   // GBK_TO_UNICODE[22068] := 16#C29A;
   // GBK_TO_UNICODE[22069] := 16#8077;
   // GBK_TO_UNICODE[22070] := 16#C29B;
   // GBK_TO_UNICODE[22071] := 16#8078;
   // GBK_TO_UNICODE[22072] := 16#C29C;
   // GBK_TO_UNICODE[22073] := 16#8079;
   // GBK_TO_UNICODE[22074] := 16#C29D;
   // GBK_TO_UNICODE[22075] := 16#807A;
   // GBK_TO_UNICODE[22076] := 16#C29E;
   // GBK_TO_UNICODE[22077] := 16#807B;
   // GBK_TO_UNICODE[22078] := 16#C29F;
   // GBK_TO_UNICODE[22079] := 16#807C;
   // GBK_TO_UNICODE[22080] := 16#C2A0;
   // GBK_TO_UNICODE[22081] := 16#807D;
   // GBK_TO_UNICODE[22082] := 16#C2A1;
   // GBK_TO_UNICODE[22083] := 16#9686;
   // GBK_TO_UNICODE[22084] := 16#C2A2;
   // GBK_TO_UNICODE[22085] := 16#5784;
   // GBK_TO_UNICODE[22086] := 16#C2A3;
   // GBK_TO_UNICODE[22087] := 16#62E2;
   // GBK_TO_UNICODE[22088] := 16#C2A4;
   // GBK_TO_UNICODE[22089] := 16#9647;
   // GBK_TO_UNICODE[22090] := 16#C2A5;
   // GBK_TO_UNICODE[22091] := 16#697C;
   // GBK_TO_UNICODE[22092] := 16#C2A6;
   // GBK_TO_UNICODE[22093] := 16#5A04;
   // GBK_TO_UNICODE[22094] := 16#C2A7;
   // GBK_TO_UNICODE[22095] := 16#6402;
   // GBK_TO_UNICODE[22096] := 16#C2A8;
   // GBK_TO_UNICODE[22097] := 16#7BD3;
   // GBK_TO_UNICODE[22098] := 16#C2A9;
   // GBK_TO_UNICODE[22099] := 16#6F0F;
   // GBK_TO_UNICODE[22100] := 16#C2AA;
   // GBK_TO_UNICODE[22101] := 16#964B;
   // GBK_TO_UNICODE[22102] := 16#C2AB;
   // GBK_TO_UNICODE[22103] := 16#82A6;
   // GBK_TO_UNICODE[22104] := 16#C2AC;
   // GBK_TO_UNICODE[22105] := 16#5362;
   // GBK_TO_UNICODE[22106] := 16#C2AD;
   // GBK_TO_UNICODE[22107] := 16#9885;
   // GBK_TO_UNICODE[22108] := 16#C2AE;
   // GBK_TO_UNICODE[22109] := 16#5E90;
   // GBK_TO_UNICODE[22110] := 16#C2AF;
   // GBK_TO_UNICODE[22111] := 16#7089;
   // GBK_TO_UNICODE[22112] := 16#C2B0;
   // GBK_TO_UNICODE[22113] := 16#63B3;
   // GBK_TO_UNICODE[22114] := 16#C2B1;
   // GBK_TO_UNICODE[22115] := 16#5364;
   // GBK_TO_UNICODE[22116] := 16#C2B2;
   // GBK_TO_UNICODE[22117] := 16#864F;
   // GBK_TO_UNICODE[22118] := 16#C2B3;
   // GBK_TO_UNICODE[22119] := 16#9C81;
   // GBK_TO_UNICODE[22120] := 16#C2B4;
   // GBK_TO_UNICODE[22121] := 16#9E93;
   // GBK_TO_UNICODE[22122] := 16#C2B5;
   // GBK_TO_UNICODE[22123] := 16#788C;
   // GBK_TO_UNICODE[22124] := 16#C2B6;
   // GBK_TO_UNICODE[22125] := 16#9732;
   // GBK_TO_UNICODE[22126] := 16#C2B7;
   // GBK_TO_UNICODE[22127] := 16#8DEF;
   // GBK_TO_UNICODE[22128] := 16#C2B8;
   // GBK_TO_UNICODE[22129] := 16#8D42;
   // GBK_TO_UNICODE[22130] := 16#C2B9;
   // GBK_TO_UNICODE[22131] := 16#9E7F;
   // GBK_TO_UNICODE[22132] := 16#C2BA;
   // GBK_TO_UNICODE[22133] := 16#6F5E;
   // GBK_TO_UNICODE[22134] := 16#C2BB;
   // GBK_TO_UNICODE[22135] := 16#7984;
   // GBK_TO_UNICODE[22136] := 16#C2BC;
   // GBK_TO_UNICODE[22137] := 16#5F55;
   // GBK_TO_UNICODE[22138] := 16#C2BD;
   // GBK_TO_UNICODE[22139] := 16#9646;
   // GBK_TO_UNICODE[22140] := 16#C2BE;
   // GBK_TO_UNICODE[22141] := 16#622E;
   // GBK_TO_UNICODE[22142] := 16#C2BF;
   // GBK_TO_UNICODE[22143] := 16#9A74;
   // GBK_TO_UNICODE[22144] := 16#C2C0;
   // GBK_TO_UNICODE[22145] := 16#5415;
   // GBK_TO_UNICODE[22146] := 16#C2C1;
   // GBK_TO_UNICODE[22147] := 16#94DD;
   // GBK_TO_UNICODE[22148] := 16#C2C2;
   // GBK_TO_UNICODE[22149] := 16#4FA3;
   // GBK_TO_UNICODE[22150] := 16#C2C3;
   // GBK_TO_UNICODE[22151] := 16#65C5;
   // GBK_TO_UNICODE[22152] := 16#C2C4;
   // GBK_TO_UNICODE[22153] := 16#5C65;
   // GBK_TO_UNICODE[22154] := 16#C2C5;
   // GBK_TO_UNICODE[22155] := 16#5C61;
   // GBK_TO_UNICODE[22156] := 16#C2C6;
   // GBK_TO_UNICODE[22157] := 16#7F15;
   // GBK_TO_UNICODE[22158] := 16#C2C7;
   // GBK_TO_UNICODE[22159] := 16#8651;
   // GBK_TO_UNICODE[22160] := 16#C2C8;
   // GBK_TO_UNICODE[22161] := 16#6C2F;
   // GBK_TO_UNICODE[22162] := 16#C2C9;
   // GBK_TO_UNICODE[22163] := 16#5F8B;
   // GBK_TO_UNICODE[22164] := 16#C2CA;
   // GBK_TO_UNICODE[22165] := 16#7387;
   // GBK_TO_UNICODE[22166] := 16#C2CB;
   // GBK_TO_UNICODE[22167] := 16#6EE4;
   // GBK_TO_UNICODE[22168] := 16#C2CC;
   // GBK_TO_UNICODE[22169] := 16#7EFF;
   // GBK_TO_UNICODE[22170] := 16#C2CD;
   // GBK_TO_UNICODE[22171] := 16#5CE6;
   // GBK_TO_UNICODE[22172] := 16#C2CE;
   // GBK_TO_UNICODE[22173] := 16#631B;
   // GBK_TO_UNICODE[22174] := 16#C2CF;
   // GBK_TO_UNICODE[22175] := 16#5B6A;
   // GBK_TO_UNICODE[22176] := 16#C2D0;
   // GBK_TO_UNICODE[22177] := 16#6EE6;
   // GBK_TO_UNICODE[22178] := 16#C2D1;
   // GBK_TO_UNICODE[22179] := 16#5375;
   // GBK_TO_UNICODE[22180] := 16#C2D2;
   // GBK_TO_UNICODE[22181] := 16#4E71;
   // GBK_TO_UNICODE[22182] := 16#C2D3;
   // GBK_TO_UNICODE[22183] := 16#63A0;
   // GBK_TO_UNICODE[22184] := 16#C2D4;
   // GBK_TO_UNICODE[22185] := 16#7565;
   // GBK_TO_UNICODE[22186] := 16#C2D5;
   // GBK_TO_UNICODE[22187] := 16#62A1;
   // GBK_TO_UNICODE[22188] := 16#C2D6;
   // GBK_TO_UNICODE[22189] := 16#8F6E;
   // GBK_TO_UNICODE[22190] := 16#C2D7;
   // GBK_TO_UNICODE[22191] := 16#4F26;
   // GBK_TO_UNICODE[22192] := 16#C2D8;
   // GBK_TO_UNICODE[22193] := 16#4ED1;
   // GBK_TO_UNICODE[22194] := 16#C2D9;
   // GBK_TO_UNICODE[22195] := 16#6CA6;
   // GBK_TO_UNICODE[22196] := 16#C2DA;
   // GBK_TO_UNICODE[22197] := 16#7EB6;
   // GBK_TO_UNICODE[22198] := 16#C2DB;
   // GBK_TO_UNICODE[22199] := 16#8BBA;
   // GBK_TO_UNICODE[22200] := 16#C2DC;
   // GBK_TO_UNICODE[22201] := 16#841D;
   // GBK_TO_UNICODE[22202] := 16#C2DD;
   // GBK_TO_UNICODE[22203] := 16#87BA;
   // GBK_TO_UNICODE[22204] := 16#C2DE;
   // GBK_TO_UNICODE[22205] := 16#7F57;
   // GBK_TO_UNICODE[22206] := 16#C2DF;
   // GBK_TO_UNICODE[22207] := 16#903B;
   // GBK_TO_UNICODE[22208] := 16#C2E0;
   // GBK_TO_UNICODE[22209] := 16#9523;
   // GBK_TO_UNICODE[22210] := 16#C2E1;
   // GBK_TO_UNICODE[22211] := 16#7BA9;
   // GBK_TO_UNICODE[22212] := 16#C2E2;
   // GBK_TO_UNICODE[22213] := 16#9AA1;
   // GBK_TO_UNICODE[22214] := 16#C2E3;
   // GBK_TO_UNICODE[22215] := 16#88F8;
   // GBK_TO_UNICODE[22216] := 16#C2E4;
   // GBK_TO_UNICODE[22217] := 16#843D;
   // GBK_TO_UNICODE[22218] := 16#C2E5;
   // GBK_TO_UNICODE[22219] := 16#6D1B;
   // GBK_TO_UNICODE[22220] := 16#C2E6;
   // GBK_TO_UNICODE[22221] := 16#9A86;
   // GBK_TO_UNICODE[22222] := 16#C2E7;
   // GBK_TO_UNICODE[22223] := 16#7EDC;
   // GBK_TO_UNICODE[22224] := 16#C2E8;
   // GBK_TO_UNICODE[22225] := 16#5988;
   // GBK_TO_UNICODE[22226] := 16#C2E9;
   // GBK_TO_UNICODE[22227] := 16#9EBB;
   // GBK_TO_UNICODE[22228] := 16#C2EA;
   // GBK_TO_UNICODE[22229] := 16#739B;
   // GBK_TO_UNICODE[22230] := 16#C2EB;
   // GBK_TO_UNICODE[22231] := 16#7801;
   // GBK_TO_UNICODE[22232] := 16#C2EC;
   // GBK_TO_UNICODE[22233] := 16#8682;
   // GBK_TO_UNICODE[22234] := 16#C2ED;
   // GBK_TO_UNICODE[22235] := 16#9A6C;
   // GBK_TO_UNICODE[22236] := 16#C2EE;
   // GBK_TO_UNICODE[22237] := 16#9A82;
   // GBK_TO_UNICODE[22238] := 16#C2EF;
   // GBK_TO_UNICODE[22239] := 16#561B;
   // GBK_TO_UNICODE[22240] := 16#C2F0;
   // GBK_TO_UNICODE[22241] := 16#5417;
   // GBK_TO_UNICODE[22242] := 16#C2F1;
   // GBK_TO_UNICODE[22243] := 16#57CB;
   // GBK_TO_UNICODE[22244] := 16#C2F2;
   // GBK_TO_UNICODE[22245] := 16#4E70;
   // GBK_TO_UNICODE[22246] := 16#C2F3;
   // GBK_TO_UNICODE[22247] := 16#9EA6;
   // GBK_TO_UNICODE[22248] := 16#C2F4;
   // GBK_TO_UNICODE[22249] := 16#5356;
   // GBK_TO_UNICODE[22250] := 16#C2F5;
   // GBK_TO_UNICODE[22251] := 16#8FC8;
   // GBK_TO_UNICODE[22252] := 16#C2F6;
   // GBK_TO_UNICODE[22253] := 16#8109;
   // GBK_TO_UNICODE[22254] := 16#C2F7;
   // GBK_TO_UNICODE[22255] := 16#7792;
   // GBK_TO_UNICODE[22256] := 16#C2F8;
   // GBK_TO_UNICODE[22257] := 16#9992;
   // GBK_TO_UNICODE[22258] := 16#C2F9;
   // GBK_TO_UNICODE[22259] := 16#86EE;
   // GBK_TO_UNICODE[22260] := 16#C2FA;
   // GBK_TO_UNICODE[22261] := 16#6EE1;
   // GBK_TO_UNICODE[22262] := 16#C2FB;
   // GBK_TO_UNICODE[22263] := 16#8513;
   // GBK_TO_UNICODE[22264] := 16#C2FC;
   // GBK_TO_UNICODE[22265] := 16#66FC;
   // GBK_TO_UNICODE[22266] := 16#C2FD;
   // GBK_TO_UNICODE[22267] := 16#6162;
   // GBK_TO_UNICODE[22268] := 16#C2FE;
   // GBK_TO_UNICODE[22269] := 16#6F2B;
   // GBK_TO_UNICODE[22270] := 16#C340;
   // GBK_TO_UNICODE[22271] := 16#807E;
   // GBK_TO_UNICODE[22272] := 16#C341;
   // GBK_TO_UNICODE[22273] := 16#8081;
   // GBK_TO_UNICODE[22274] := 16#C342;
   // GBK_TO_UNICODE[22275] := 16#8082;
   // GBK_TO_UNICODE[22276] := 16#C343;
   // GBK_TO_UNICODE[22277] := 16#8085;
   // GBK_TO_UNICODE[22278] := 16#C344;
   // GBK_TO_UNICODE[22279] := 16#8088;
   // GBK_TO_UNICODE[22280] := 16#C345;
   // GBK_TO_UNICODE[22281] := 16#808A;
   // GBK_TO_UNICODE[22282] := 16#C346;
   // GBK_TO_UNICODE[22283] := 16#808D;
   // GBK_TO_UNICODE[22284] := 16#C347;
   // GBK_TO_UNICODE[22285] := 16#808E;
   // GBK_TO_UNICODE[22286] := 16#C348;
   // GBK_TO_UNICODE[22287] := 16#808F;
   // GBK_TO_UNICODE[22288] := 16#C349;
   // GBK_TO_UNICODE[22289] := 16#8090;
   // GBK_TO_UNICODE[22290] := 16#C34A;
   // GBK_TO_UNICODE[22291] := 16#8091;
   // GBK_TO_UNICODE[22292] := 16#C34B;
   // GBK_TO_UNICODE[22293] := 16#8092;
   // GBK_TO_UNICODE[22294] := 16#C34C;
   // GBK_TO_UNICODE[22295] := 16#8094;
   // GBK_TO_UNICODE[22296] := 16#C34D;
   // GBK_TO_UNICODE[22297] := 16#8095;
   // GBK_TO_UNICODE[22298] := 16#C34E;
   // GBK_TO_UNICODE[22299] := 16#8097;
   // GBK_TO_UNICODE[22300] := 16#C34F;
   // GBK_TO_UNICODE[22301] := 16#8099;
   // GBK_TO_UNICODE[22302] := 16#C350;
   // GBK_TO_UNICODE[22303] := 16#809E;
   // GBK_TO_UNICODE[22304] := 16#C351;
   // GBK_TO_UNICODE[22305] := 16#80A3;
   // GBK_TO_UNICODE[22306] := 16#C352;
   // GBK_TO_UNICODE[22307] := 16#80A6;
   // GBK_TO_UNICODE[22308] := 16#C353;
   // GBK_TO_UNICODE[22309] := 16#80A7;
   // GBK_TO_UNICODE[22310] := 16#C354;
   // GBK_TO_UNICODE[22311] := 16#80A8;
   // GBK_TO_UNICODE[22312] := 16#C355;
   // GBK_TO_UNICODE[22313] := 16#80AC;
   // GBK_TO_UNICODE[22314] := 16#C356;
   // GBK_TO_UNICODE[22315] := 16#80B0;
   // GBK_TO_UNICODE[22316] := 16#C357;
   // GBK_TO_UNICODE[22317] := 16#80B3;
   // GBK_TO_UNICODE[22318] := 16#C358;
   // GBK_TO_UNICODE[22319] := 16#80B5;
   // GBK_TO_UNICODE[22320] := 16#C359;
   // GBK_TO_UNICODE[22321] := 16#80B6;
   // GBK_TO_UNICODE[22322] := 16#C35A;
   // GBK_TO_UNICODE[22323] := 16#80B8;
   // GBK_TO_UNICODE[22324] := 16#C35B;
   // GBK_TO_UNICODE[22325] := 16#80B9;
   // GBK_TO_UNICODE[22326] := 16#C35C;
   // GBK_TO_UNICODE[22327] := 16#80BB;
   // GBK_TO_UNICODE[22328] := 16#C35D;
   // GBK_TO_UNICODE[22329] := 16#80C5;
   // GBK_TO_UNICODE[22330] := 16#C35E;
   // GBK_TO_UNICODE[22331] := 16#80C7;
   // GBK_TO_UNICODE[22332] := 16#C35F;
   // GBK_TO_UNICODE[22333] := 16#80C8;
   // GBK_TO_UNICODE[22334] := 16#C360;
   // GBK_TO_UNICODE[22335] := 16#80C9;
   // GBK_TO_UNICODE[22336] := 16#C361;
   // GBK_TO_UNICODE[22337] := 16#80CA;
   // GBK_TO_UNICODE[22338] := 16#C362;
   // GBK_TO_UNICODE[22339] := 16#80CB;
   // GBK_TO_UNICODE[22340] := 16#C363;
   // GBK_TO_UNICODE[22341] := 16#80CF;
   // GBK_TO_UNICODE[22342] := 16#C364;
   // GBK_TO_UNICODE[22343] := 16#80D0;
   // GBK_TO_UNICODE[22344] := 16#C365;
   // GBK_TO_UNICODE[22345] := 16#80D1;
   // GBK_TO_UNICODE[22346] := 16#C366;
   // GBK_TO_UNICODE[22347] := 16#80D2;
   // GBK_TO_UNICODE[22348] := 16#C367;
   // GBK_TO_UNICODE[22349] := 16#80D3;
   // GBK_TO_UNICODE[22350] := 16#C368;
   // GBK_TO_UNICODE[22351] := 16#80D4;
   // GBK_TO_UNICODE[22352] := 16#C369;
   // GBK_TO_UNICODE[22353] := 16#80D5;
   // GBK_TO_UNICODE[22354] := 16#C36A;
   // GBK_TO_UNICODE[22355] := 16#80D8;
   // GBK_TO_UNICODE[22356] := 16#C36B;
   // GBK_TO_UNICODE[22357] := 16#80DF;
   // GBK_TO_UNICODE[22358] := 16#C36C;
   // GBK_TO_UNICODE[22359] := 16#80E0;
   // GBK_TO_UNICODE[22360] := 16#C36D;
   // GBK_TO_UNICODE[22361] := 16#80E2;
   // GBK_TO_UNICODE[22362] := 16#C36E;
   // GBK_TO_UNICODE[22363] := 16#80E3;
   // GBK_TO_UNICODE[22364] := 16#C36F;
   // GBK_TO_UNICODE[22365] := 16#80E6;
   // GBK_TO_UNICODE[22366] := 16#C370;
   // GBK_TO_UNICODE[22367] := 16#80EE;
   // GBK_TO_UNICODE[22368] := 16#C371;
   // GBK_TO_UNICODE[22369] := 16#80F5;
   // GBK_TO_UNICODE[22370] := 16#C372;
   // GBK_TO_UNICODE[22371] := 16#80F7;
   // GBK_TO_UNICODE[22372] := 16#C373;
   // GBK_TO_UNICODE[22373] := 16#80F9;
   // GBK_TO_UNICODE[22374] := 16#C374;
   // GBK_TO_UNICODE[22375] := 16#80FB;
   // GBK_TO_UNICODE[22376] := 16#C375;
   // GBK_TO_UNICODE[22377] := 16#80FE;
   // GBK_TO_UNICODE[22378] := 16#C376;
   // GBK_TO_UNICODE[22379] := 16#80FF;
   // GBK_TO_UNICODE[22380] := 16#C377;
   // GBK_TO_UNICODE[22381] := 16#8100;
   // GBK_TO_UNICODE[22382] := 16#C378;
   // GBK_TO_UNICODE[22383] := 16#8101;
   // GBK_TO_UNICODE[22384] := 16#C379;
   // GBK_TO_UNICODE[22385] := 16#8103;
   // GBK_TO_UNICODE[22386] := 16#C37A;
   // GBK_TO_UNICODE[22387] := 16#8104;
   // GBK_TO_UNICODE[22388] := 16#C37B;
   // GBK_TO_UNICODE[22389] := 16#8105;
   // GBK_TO_UNICODE[22390] := 16#C37C;
   // GBK_TO_UNICODE[22391] := 16#8107;
   // GBK_TO_UNICODE[22392] := 16#C37D;
   // GBK_TO_UNICODE[22393] := 16#8108;
   // GBK_TO_UNICODE[22394] := 16#C37E;
   // GBK_TO_UNICODE[22395] := 16#810B;
   // GBK_TO_UNICODE[22396] := 16#C380;
   // GBK_TO_UNICODE[22397] := 16#810C;
   // GBK_TO_UNICODE[22398] := 16#C381;
   // GBK_TO_UNICODE[22399] := 16#8115;
   // GBK_TO_UNICODE[22400] := 16#C382;
   // GBK_TO_UNICODE[22401] := 16#8117;
   // GBK_TO_UNICODE[22402] := 16#C383;
   // GBK_TO_UNICODE[22403] := 16#8119;
   // GBK_TO_UNICODE[22404] := 16#C384;
   // GBK_TO_UNICODE[22405] := 16#811B;
   // GBK_TO_UNICODE[22406] := 16#C385;
   // GBK_TO_UNICODE[22407] := 16#811C;
   // GBK_TO_UNICODE[22408] := 16#C386;
   // GBK_TO_UNICODE[22409] := 16#811D;
   // GBK_TO_UNICODE[22410] := 16#C387;
   // GBK_TO_UNICODE[22411] := 16#811F;
   // GBK_TO_UNICODE[22412] := 16#C388;
   // GBK_TO_UNICODE[22413] := 16#8120;
   // GBK_TO_UNICODE[22414] := 16#C389;
   // GBK_TO_UNICODE[22415] := 16#8121;
   // GBK_TO_UNICODE[22416] := 16#C38A;
   // GBK_TO_UNICODE[22417] := 16#8122;
   // GBK_TO_UNICODE[22418] := 16#C38B;
   // GBK_TO_UNICODE[22419] := 16#8123;
   // GBK_TO_UNICODE[22420] := 16#C38C;
   // GBK_TO_UNICODE[22421] := 16#8124;
   // GBK_TO_UNICODE[22422] := 16#C38D;
   // GBK_TO_UNICODE[22423] := 16#8125;
   // GBK_TO_UNICODE[22424] := 16#C38E;
   // GBK_TO_UNICODE[22425] := 16#8126;
   // GBK_TO_UNICODE[22426] := 16#C38F;
   // GBK_TO_UNICODE[22427] := 16#8127;
   // GBK_TO_UNICODE[22428] := 16#C390;
   // GBK_TO_UNICODE[22429] := 16#8128;
   // GBK_TO_UNICODE[22430] := 16#C391;
   // GBK_TO_UNICODE[22431] := 16#8129;
   // GBK_TO_UNICODE[22432] := 16#C392;
   // GBK_TO_UNICODE[22433] := 16#812A;
   // GBK_TO_UNICODE[22434] := 16#C393;
   // GBK_TO_UNICODE[22435] := 16#812B;
   // GBK_TO_UNICODE[22436] := 16#C394;
   // GBK_TO_UNICODE[22437] := 16#812D;
   // GBK_TO_UNICODE[22438] := 16#C395;
   // GBK_TO_UNICODE[22439] := 16#812E;
   // GBK_TO_UNICODE[22440] := 16#C396;
   // GBK_TO_UNICODE[22441] := 16#8130;
   // GBK_TO_UNICODE[22442] := 16#C397;
   // GBK_TO_UNICODE[22443] := 16#8133;
   // GBK_TO_UNICODE[22444] := 16#C398;
   // GBK_TO_UNICODE[22445] := 16#8134;
   // GBK_TO_UNICODE[22446] := 16#C399;
   // GBK_TO_UNICODE[22447] := 16#8135;
   // GBK_TO_UNICODE[22448] := 16#C39A;
   // GBK_TO_UNICODE[22449] := 16#8137;
   // GBK_TO_UNICODE[22450] := 16#C39B;
   // GBK_TO_UNICODE[22451] := 16#8139;
   // GBK_TO_UNICODE[22452] := 16#C39C;
   // GBK_TO_UNICODE[22453] := 16#813A;
   // GBK_TO_UNICODE[22454] := 16#C39D;
   // GBK_TO_UNICODE[22455] := 16#813B;
   // GBK_TO_UNICODE[22456] := 16#C39E;
   // GBK_TO_UNICODE[22457] := 16#813C;
   // GBK_TO_UNICODE[22458] := 16#C39F;
   // GBK_TO_UNICODE[22459] := 16#813D;
   // GBK_TO_UNICODE[22460] := 16#C3A0;
   // GBK_TO_UNICODE[22461] := 16#813F;
   // GBK_TO_UNICODE[22462] := 16#C3A1;
   // GBK_TO_UNICODE[22463] := 16#8C29;
   // GBK_TO_UNICODE[22464] := 16#C3A2;
   // GBK_TO_UNICODE[22465] := 16#8292;
   // GBK_TO_UNICODE[22466] := 16#C3A3;
   // GBK_TO_UNICODE[22467] := 16#832B;
   // GBK_TO_UNICODE[22468] := 16#C3A4;
   // GBK_TO_UNICODE[22469] := 16#76F2;
   // GBK_TO_UNICODE[22470] := 16#C3A5;
   // GBK_TO_UNICODE[22471] := 16#6C13;
   // GBK_TO_UNICODE[22472] := 16#C3A6;
   // GBK_TO_UNICODE[22473] := 16#5FD9;
   // GBK_TO_UNICODE[22474] := 16#C3A7;
   // GBK_TO_UNICODE[22475] := 16#83BD;
   // GBK_TO_UNICODE[22476] := 16#C3A8;
   // GBK_TO_UNICODE[22477] := 16#732B;
   // GBK_TO_UNICODE[22478] := 16#C3A9;
   // GBK_TO_UNICODE[22479] := 16#8305;
   // GBK_TO_UNICODE[22480] := 16#C3AA;
   // GBK_TO_UNICODE[22481] := 16#951A;
   // GBK_TO_UNICODE[22482] := 16#C3AB;
   // GBK_TO_UNICODE[22483] := 16#6BDB;
   // GBK_TO_UNICODE[22484] := 16#C3AC;
   // GBK_TO_UNICODE[22485] := 16#77DB;
   // GBK_TO_UNICODE[22486] := 16#C3AD;
   // GBK_TO_UNICODE[22487] := 16#94C6;
   // GBK_TO_UNICODE[22488] := 16#C3AE;
   // GBK_TO_UNICODE[22489] := 16#536F;
   // GBK_TO_UNICODE[22490] := 16#C3AF;
   // GBK_TO_UNICODE[22491] := 16#8302;
   // GBK_TO_UNICODE[22492] := 16#C3B0;
   // GBK_TO_UNICODE[22493] := 16#5192;
   // GBK_TO_UNICODE[22494] := 16#C3B1;
   // GBK_TO_UNICODE[22495] := 16#5E3D;
   // GBK_TO_UNICODE[22496] := 16#C3B2;
   // GBK_TO_UNICODE[22497] := 16#8C8C;
   // GBK_TO_UNICODE[22498] := 16#C3B3;
   // GBK_TO_UNICODE[22499] := 16#8D38;
   // GBK_TO_UNICODE[22500] := 16#C3B4;
   // GBK_TO_UNICODE[22501] := 16#4E48;
   // GBK_TO_UNICODE[22502] := 16#C3B5;
   // GBK_TO_UNICODE[22503] := 16#73AB;
   // GBK_TO_UNICODE[22504] := 16#C3B6;
   // GBK_TO_UNICODE[22505] := 16#679A;
   // GBK_TO_UNICODE[22506] := 16#C3B7;
   // GBK_TO_UNICODE[22507] := 16#6885;
   // GBK_TO_UNICODE[22508] := 16#C3B8;
   // GBK_TO_UNICODE[22509] := 16#9176;
   // GBK_TO_UNICODE[22510] := 16#C3B9;
   // GBK_TO_UNICODE[22511] := 16#9709;
   // GBK_TO_UNICODE[22512] := 16#C3BA;
   // GBK_TO_UNICODE[22513] := 16#7164;
   // GBK_TO_UNICODE[22514] := 16#C3BB;
   // GBK_TO_UNICODE[22515] := 16#6CA1;
   // GBK_TO_UNICODE[22516] := 16#C3BC;
   // GBK_TO_UNICODE[22517] := 16#7709;
   // GBK_TO_UNICODE[22518] := 16#C3BD;
   // GBK_TO_UNICODE[22519] := 16#5A92;
   // GBK_TO_UNICODE[22520] := 16#C3BE;
   // GBK_TO_UNICODE[22521] := 16#9541;
   // GBK_TO_UNICODE[22522] := 16#C3BF;
   // GBK_TO_UNICODE[22523] := 16#6BCF;
   // GBK_TO_UNICODE[22524] := 16#C3C0;
   // GBK_TO_UNICODE[22525] := 16#7F8E;
   // GBK_TO_UNICODE[22526] := 16#C3C1;
   // GBK_TO_UNICODE[22527] := 16#6627;
   // GBK_TO_UNICODE[22528] := 16#C3C2;
   // GBK_TO_UNICODE[22529] := 16#5BD0;
   // GBK_TO_UNICODE[22530] := 16#C3C3;
   // GBK_TO_UNICODE[22531] := 16#59B9;
   // GBK_TO_UNICODE[22532] := 16#C3C4;
   // GBK_TO_UNICODE[22533] := 16#5A9A;
   // GBK_TO_UNICODE[22534] := 16#C3C5;
   // GBK_TO_UNICODE[22535] := 16#95E8;
   // GBK_TO_UNICODE[22536] := 16#C3C6;
   // GBK_TO_UNICODE[22537] := 16#95F7;
   // GBK_TO_UNICODE[22538] := 16#C3C7;
   // GBK_TO_UNICODE[22539] := 16#4EEC;
   // GBK_TO_UNICODE[22540] := 16#C3C8;
   // GBK_TO_UNICODE[22541] := 16#840C;
   // GBK_TO_UNICODE[22542] := 16#C3C9;
   // GBK_TO_UNICODE[22543] := 16#8499;
   // GBK_TO_UNICODE[22544] := 16#C3CA;
   // GBK_TO_UNICODE[22545] := 16#6AAC;
   // GBK_TO_UNICODE[22546] := 16#C3CB;
   // GBK_TO_UNICODE[22547] := 16#76DF;
   // GBK_TO_UNICODE[22548] := 16#C3CC;
   // GBK_TO_UNICODE[22549] := 16#9530;
   // GBK_TO_UNICODE[22550] := 16#C3CD;
   // GBK_TO_UNICODE[22551] := 16#731B;
   // GBK_TO_UNICODE[22552] := 16#C3CE;
   // GBK_TO_UNICODE[22553] := 16#68A6;
   // GBK_TO_UNICODE[22554] := 16#C3CF;
   // GBK_TO_UNICODE[22555] := 16#5B5F;
   // GBK_TO_UNICODE[22556] := 16#C3D0;
   // GBK_TO_UNICODE[22557] := 16#772F;
   // GBK_TO_UNICODE[22558] := 16#C3D1;
   // GBK_TO_UNICODE[22559] := 16#919A;
   // GBK_TO_UNICODE[22560] := 16#C3D2;
   // GBK_TO_UNICODE[22561] := 16#9761;
   // GBK_TO_UNICODE[22562] := 16#C3D3;
   // GBK_TO_UNICODE[22563] := 16#7CDC;
   // GBK_TO_UNICODE[22564] := 16#C3D4;
   // GBK_TO_UNICODE[22565] := 16#8FF7;
   // GBK_TO_UNICODE[22566] := 16#C3D5;
   // GBK_TO_UNICODE[22567] := 16#8C1C;
   // GBK_TO_UNICODE[22568] := 16#C3D6;
   // GBK_TO_UNICODE[22569] := 16#5F25;
   // GBK_TO_UNICODE[22570] := 16#C3D7;
   // GBK_TO_UNICODE[22571] := 16#7C73;
   // GBK_TO_UNICODE[22572] := 16#C3D8;
   // GBK_TO_UNICODE[22573] := 16#79D8;
   // GBK_TO_UNICODE[22574] := 16#C3D9;
   // GBK_TO_UNICODE[22575] := 16#89C5;
   // GBK_TO_UNICODE[22576] := 16#C3DA;
   // GBK_TO_UNICODE[22577] := 16#6CCC;
   // GBK_TO_UNICODE[22578] := 16#C3DB;
   // GBK_TO_UNICODE[22579] := 16#871C;
   // GBK_TO_UNICODE[22580] := 16#C3DC;
   // GBK_TO_UNICODE[22581] := 16#5BC6;
   // GBK_TO_UNICODE[22582] := 16#C3DD;
   // GBK_TO_UNICODE[22583] := 16#5E42;
   // GBK_TO_UNICODE[22584] := 16#C3DE;
   // GBK_TO_UNICODE[22585] := 16#68C9;
   // GBK_TO_UNICODE[22586] := 16#C3DF;
   // GBK_TO_UNICODE[22587] := 16#7720;
   // GBK_TO_UNICODE[22588] := 16#C3E0;
   // GBK_TO_UNICODE[22589] := 16#7EF5;
   // GBK_TO_UNICODE[22590] := 16#C3E1;
   // GBK_TO_UNICODE[22591] := 16#5195;
   // GBK_TO_UNICODE[22592] := 16#C3E2;
   // GBK_TO_UNICODE[22593] := 16#514D;
   // GBK_TO_UNICODE[22594] := 16#C3E3;
   // GBK_TO_UNICODE[22595] := 16#52C9;
   // GBK_TO_UNICODE[22596] := 16#C3E4;
   // GBK_TO_UNICODE[22597] := 16#5A29;
   // GBK_TO_UNICODE[22598] := 16#C3E5;
   // GBK_TO_UNICODE[22599] := 16#7F05;
   // GBK_TO_UNICODE[22600] := 16#C3E6;
   // GBK_TO_UNICODE[22601] := 16#9762;
   // GBK_TO_UNICODE[22602] := 16#C3E7;
   // GBK_TO_UNICODE[22603] := 16#82D7;
   // GBK_TO_UNICODE[22604] := 16#C3E8;
   // GBK_TO_UNICODE[22605] := 16#63CF;
   // GBK_TO_UNICODE[22606] := 16#C3E9;
   // GBK_TO_UNICODE[22607] := 16#7784;
   // GBK_TO_UNICODE[22608] := 16#C3EA;
   // GBK_TO_UNICODE[22609] := 16#85D0;
   // GBK_TO_UNICODE[22610] := 16#C3EB;
   // GBK_TO_UNICODE[22611] := 16#79D2;
   // GBK_TO_UNICODE[22612] := 16#C3EC;
   // GBK_TO_UNICODE[22613] := 16#6E3A;
   // GBK_TO_UNICODE[22614] := 16#C3ED;
   // GBK_TO_UNICODE[22615] := 16#5E99;
   // GBK_TO_UNICODE[22616] := 16#C3EE;
   // GBK_TO_UNICODE[22617] := 16#5999;
   // GBK_TO_UNICODE[22618] := 16#C3EF;
   // GBK_TO_UNICODE[22619] := 16#8511;
   // GBK_TO_UNICODE[22620] := 16#C3F0;
   // GBK_TO_UNICODE[22621] := 16#706D;
   // GBK_TO_UNICODE[22622] := 16#C3F1;
   // GBK_TO_UNICODE[22623] := 16#6C11;
   // GBK_TO_UNICODE[22624] := 16#C3F2;
   // GBK_TO_UNICODE[22625] := 16#62BF;
   // GBK_TO_UNICODE[22626] := 16#C3F3;
   // GBK_TO_UNICODE[22627] := 16#76BF;
   // GBK_TO_UNICODE[22628] := 16#C3F4;
   // GBK_TO_UNICODE[22629] := 16#654F;
   // GBK_TO_UNICODE[22630] := 16#C3F5;
   // GBK_TO_UNICODE[22631] := 16#60AF;
   // GBK_TO_UNICODE[22632] := 16#C3F6;
   // GBK_TO_UNICODE[22633] := 16#95FD;
   // GBK_TO_UNICODE[22634] := 16#C3F7;
   // GBK_TO_UNICODE[22635] := 16#660E;
   // GBK_TO_UNICODE[22636] := 16#C3F8;
   // GBK_TO_UNICODE[22637] := 16#879F;
   // GBK_TO_UNICODE[22638] := 16#C3F9;
   // GBK_TO_UNICODE[22639] := 16#9E23;
   // GBK_TO_UNICODE[22640] := 16#C3FA;
   // GBK_TO_UNICODE[22641] := 16#94ED;
   // GBK_TO_UNICODE[22642] := 16#C3FB;
   // GBK_TO_UNICODE[22643] := 16#540D;
   // GBK_TO_UNICODE[22644] := 16#C3FC;
   // GBK_TO_UNICODE[22645] := 16#547D;
   // GBK_TO_UNICODE[22646] := 16#C3FD;
   // GBK_TO_UNICODE[22647] := 16#8C2C;
   // GBK_TO_UNICODE[22648] := 16#C3FE;
   // GBK_TO_UNICODE[22649] := 16#6478;
   // GBK_TO_UNICODE[22650] := 16#C440;
   // GBK_TO_UNICODE[22651] := 16#8140;
   // GBK_TO_UNICODE[22652] := 16#C441;
   // GBK_TO_UNICODE[22653] := 16#8141;
   // GBK_TO_UNICODE[22654] := 16#C442;
   // GBK_TO_UNICODE[22655] := 16#8142;
   // GBK_TO_UNICODE[22656] := 16#C443;
   // GBK_TO_UNICODE[22657] := 16#8143;
   // GBK_TO_UNICODE[22658] := 16#C444;
   // GBK_TO_UNICODE[22659] := 16#8144;
   // GBK_TO_UNICODE[22660] := 16#C445;
   // GBK_TO_UNICODE[22661] := 16#8145;
   // GBK_TO_UNICODE[22662] := 16#C446;
   // GBK_TO_UNICODE[22663] := 16#8147;
   // GBK_TO_UNICODE[22664] := 16#C447;
   // GBK_TO_UNICODE[22665] := 16#8149;
   // GBK_TO_UNICODE[22666] := 16#C448;
   // GBK_TO_UNICODE[22667] := 16#814D;
   // GBK_TO_UNICODE[22668] := 16#C449;
   // GBK_TO_UNICODE[22669] := 16#814E;
   // GBK_TO_UNICODE[22670] := 16#C44A;
   // GBK_TO_UNICODE[22671] := 16#814F;
   // GBK_TO_UNICODE[22672] := 16#C44B;
   // GBK_TO_UNICODE[22673] := 16#8152;
   // GBK_TO_UNICODE[22674] := 16#C44C;
   // GBK_TO_UNICODE[22675] := 16#8156;
   // GBK_TO_UNICODE[22676] := 16#C44D;
   // GBK_TO_UNICODE[22677] := 16#8157;
   // GBK_TO_UNICODE[22678] := 16#C44E;
   // GBK_TO_UNICODE[22679] := 16#8158;
   // GBK_TO_UNICODE[22680] := 16#C44F;
   // GBK_TO_UNICODE[22681] := 16#815B;
   // GBK_TO_UNICODE[22682] := 16#C450;
   // GBK_TO_UNICODE[22683] := 16#815C;
   // GBK_TO_UNICODE[22684] := 16#C451;
   // GBK_TO_UNICODE[22685] := 16#815D;
   // GBK_TO_UNICODE[22686] := 16#C452;
   // GBK_TO_UNICODE[22687] := 16#815E;
   // GBK_TO_UNICODE[22688] := 16#C453;
   // GBK_TO_UNICODE[22689] := 16#815F;
   // GBK_TO_UNICODE[22690] := 16#C454;
   // GBK_TO_UNICODE[22691] := 16#8161;
   // GBK_TO_UNICODE[22692] := 16#C455;
   // GBK_TO_UNICODE[22693] := 16#8162;
   // GBK_TO_UNICODE[22694] := 16#C456;
   // GBK_TO_UNICODE[22695] := 16#8163;
   // GBK_TO_UNICODE[22696] := 16#C457;
   // GBK_TO_UNICODE[22697] := 16#8164;
   // GBK_TO_UNICODE[22698] := 16#C458;
   // GBK_TO_UNICODE[22699] := 16#8166;
   // GBK_TO_UNICODE[22700] := 16#C459;
   // GBK_TO_UNICODE[22701] := 16#8168;
   // GBK_TO_UNICODE[22702] := 16#C45A;
   // GBK_TO_UNICODE[22703] := 16#816A;
   // GBK_TO_UNICODE[22704] := 16#C45B;
   // GBK_TO_UNICODE[22705] := 16#816B;
   // GBK_TO_UNICODE[22706] := 16#C45C;
   // GBK_TO_UNICODE[22707] := 16#816C;
   // GBK_TO_UNICODE[22708] := 16#C45D;
   // GBK_TO_UNICODE[22709] := 16#816F;
   // GBK_TO_UNICODE[22710] := 16#C45E;
   // GBK_TO_UNICODE[22711] := 16#8172;
   // GBK_TO_UNICODE[22712] := 16#C45F;
   // GBK_TO_UNICODE[22713] := 16#8173;
   // GBK_TO_UNICODE[22714] := 16#C460;
   // GBK_TO_UNICODE[22715] := 16#8175;
   // GBK_TO_UNICODE[22716] := 16#C461;
   // GBK_TO_UNICODE[22717] := 16#8176;
   // GBK_TO_UNICODE[22718] := 16#C462;
   // GBK_TO_UNICODE[22719] := 16#8177;
   // GBK_TO_UNICODE[22720] := 16#C463;
   // GBK_TO_UNICODE[22721] := 16#8178;
   // GBK_TO_UNICODE[22722] := 16#C464;
   // GBK_TO_UNICODE[22723] := 16#8181;
   // GBK_TO_UNICODE[22724] := 16#C465;
   // GBK_TO_UNICODE[22725] := 16#8183;
   // GBK_TO_UNICODE[22726] := 16#C466;
   // GBK_TO_UNICODE[22727] := 16#8184;
   // GBK_TO_UNICODE[22728] := 16#C467;
   // GBK_TO_UNICODE[22729] := 16#8185;
   // GBK_TO_UNICODE[22730] := 16#C468;
   // GBK_TO_UNICODE[22731] := 16#8186;
   // GBK_TO_UNICODE[22732] := 16#C469;
   // GBK_TO_UNICODE[22733] := 16#8187;
   // GBK_TO_UNICODE[22734] := 16#C46A;
   // GBK_TO_UNICODE[22735] := 16#8189;
   // GBK_TO_UNICODE[22736] := 16#C46B;
   // GBK_TO_UNICODE[22737] := 16#818B;
   // GBK_TO_UNICODE[22738] := 16#C46C;
   // GBK_TO_UNICODE[22739] := 16#818C;
   // GBK_TO_UNICODE[22740] := 16#C46D;
   // GBK_TO_UNICODE[22741] := 16#818D;
   // GBK_TO_UNICODE[22742] := 16#C46E;
   // GBK_TO_UNICODE[22743] := 16#818E;
   // GBK_TO_UNICODE[22744] := 16#C46F;
   // GBK_TO_UNICODE[22745] := 16#8190;
   // GBK_TO_UNICODE[22746] := 16#C470;
   // GBK_TO_UNICODE[22747] := 16#8192;
   // GBK_TO_UNICODE[22748] := 16#C471;
   // GBK_TO_UNICODE[22749] := 16#8193;
   // GBK_TO_UNICODE[22750] := 16#C472;
   // GBK_TO_UNICODE[22751] := 16#8194;
   // GBK_TO_UNICODE[22752] := 16#C473;
   // GBK_TO_UNICODE[22753] := 16#8195;
   // GBK_TO_UNICODE[22754] := 16#C474;
   // GBK_TO_UNICODE[22755] := 16#8196;
   // GBK_TO_UNICODE[22756] := 16#C475;
   // GBK_TO_UNICODE[22757] := 16#8197;
   // GBK_TO_UNICODE[22758] := 16#C476;
   // GBK_TO_UNICODE[22759] := 16#8199;
   // GBK_TO_UNICODE[22760] := 16#C477;
   // GBK_TO_UNICODE[22761] := 16#819A;
   // GBK_TO_UNICODE[22762] := 16#C478;
   // GBK_TO_UNICODE[22763] := 16#819E;
   // GBK_TO_UNICODE[22764] := 16#C479;
   // GBK_TO_UNICODE[22765] := 16#819F;
   // GBK_TO_UNICODE[22766] := 16#C47A;
   // GBK_TO_UNICODE[22767] := 16#81A0;
   // GBK_TO_UNICODE[22768] := 16#C47B;
   // GBK_TO_UNICODE[22769] := 16#81A1;
   // GBK_TO_UNICODE[22770] := 16#C47C;
   // GBK_TO_UNICODE[22771] := 16#81A2;
   // GBK_TO_UNICODE[22772] := 16#C47D;
   // GBK_TO_UNICODE[22773] := 16#81A4;
   // GBK_TO_UNICODE[22774] := 16#C47E;
   // GBK_TO_UNICODE[22775] := 16#81A5;
   // GBK_TO_UNICODE[22776] := 16#C480;
   // GBK_TO_UNICODE[22777] := 16#81A7;
   // GBK_TO_UNICODE[22778] := 16#C481;
   // GBK_TO_UNICODE[22779] := 16#81A9;
   // GBK_TO_UNICODE[22780] := 16#C482;
   // GBK_TO_UNICODE[22781] := 16#81AB;
   // GBK_TO_UNICODE[22782] := 16#C483;
   // GBK_TO_UNICODE[22783] := 16#81AC;
   // GBK_TO_UNICODE[22784] := 16#C484;
   // GBK_TO_UNICODE[22785] := 16#81AD;
   // GBK_TO_UNICODE[22786] := 16#C485;
   // GBK_TO_UNICODE[22787] := 16#81AE;
   // GBK_TO_UNICODE[22788] := 16#C486;
   // GBK_TO_UNICODE[22789] := 16#81AF;
   // GBK_TO_UNICODE[22790] := 16#C487;
   // GBK_TO_UNICODE[22791] := 16#81B0;
   // GBK_TO_UNICODE[22792] := 16#C488;
   // GBK_TO_UNICODE[22793] := 16#81B1;
   // GBK_TO_UNICODE[22794] := 16#C489;
   // GBK_TO_UNICODE[22795] := 16#81B2;
   // GBK_TO_UNICODE[22796] := 16#C48A;
   // GBK_TO_UNICODE[22797] := 16#81B4;
   // GBK_TO_UNICODE[22798] := 16#C48B;
   // GBK_TO_UNICODE[22799] := 16#81B5;
   // GBK_TO_UNICODE[22800] := 16#C48C;
   // GBK_TO_UNICODE[22801] := 16#81B6;
   // GBK_TO_UNICODE[22802] := 16#C48D;
   // GBK_TO_UNICODE[22803] := 16#81B7;
   // GBK_TO_UNICODE[22804] := 16#C48E;
   // GBK_TO_UNICODE[22805] := 16#81B8;
   // GBK_TO_UNICODE[22806] := 16#C48F;
   // GBK_TO_UNICODE[22807] := 16#81B9;
   // GBK_TO_UNICODE[22808] := 16#C490;
   // GBK_TO_UNICODE[22809] := 16#81BC;
   // GBK_TO_UNICODE[22810] := 16#C491;
   // GBK_TO_UNICODE[22811] := 16#81BD;
   // GBK_TO_UNICODE[22812] := 16#C492;
   // GBK_TO_UNICODE[22813] := 16#81BE;
   // GBK_TO_UNICODE[22814] := 16#C493;
   // GBK_TO_UNICODE[22815] := 16#81BF;
   // GBK_TO_UNICODE[22816] := 16#C494;
   // GBK_TO_UNICODE[22817] := 16#81C4;
   // GBK_TO_UNICODE[22818] := 16#C495;
   // GBK_TO_UNICODE[22819] := 16#81C5;
   // GBK_TO_UNICODE[22820] := 16#C496;
   // GBK_TO_UNICODE[22821] := 16#81C7;
   // GBK_TO_UNICODE[22822] := 16#C497;
   // GBK_TO_UNICODE[22823] := 16#81C8;
   // GBK_TO_UNICODE[22824] := 16#C498;
   // GBK_TO_UNICODE[22825] := 16#81C9;
   // GBK_TO_UNICODE[22826] := 16#C499;
   // GBK_TO_UNICODE[22827] := 16#81CB;
   // GBK_TO_UNICODE[22828] := 16#C49A;
   // GBK_TO_UNICODE[22829] := 16#81CD;
   // GBK_TO_UNICODE[22830] := 16#C49B;
   // GBK_TO_UNICODE[22831] := 16#81CE;
   // GBK_TO_UNICODE[22832] := 16#C49C;
   // GBK_TO_UNICODE[22833] := 16#81CF;
   // GBK_TO_UNICODE[22834] := 16#C49D;
   // GBK_TO_UNICODE[22835] := 16#81D0;
   // GBK_TO_UNICODE[22836] := 16#C49E;
   // GBK_TO_UNICODE[22837] := 16#81D1;
   // GBK_TO_UNICODE[22838] := 16#C49F;
   // GBK_TO_UNICODE[22839] := 16#81D2;
   // GBK_TO_UNICODE[22840] := 16#C4A0;
   // GBK_TO_UNICODE[22841] := 16#81D3;
   // GBK_TO_UNICODE[22842] := 16#C4A1;
   // GBK_TO_UNICODE[22843] := 16#6479;
   // GBK_TO_UNICODE[22844] := 16#C4A2;
   // GBK_TO_UNICODE[22845] := 16#8611;
   // GBK_TO_UNICODE[22846] := 16#C4A3;
   // GBK_TO_UNICODE[22847] := 16#6A21;
   // GBK_TO_UNICODE[22848] := 16#C4A4;
   // GBK_TO_UNICODE[22849] := 16#819C;
   // GBK_TO_UNICODE[22850] := 16#C4A5;
   // GBK_TO_UNICODE[22851] := 16#78E8;
   // GBK_TO_UNICODE[22852] := 16#C4A6;
   // GBK_TO_UNICODE[22853] := 16#6469;
   // GBK_TO_UNICODE[22854] := 16#C4A7;
   // GBK_TO_UNICODE[22855] := 16#9B54;
   // GBK_TO_UNICODE[22856] := 16#C4A8;
   // GBK_TO_UNICODE[22857] := 16#62B9;
   // GBK_TO_UNICODE[22858] := 16#C4A9;
   // GBK_TO_UNICODE[22859] := 16#672B;
   // GBK_TO_UNICODE[22860] := 16#C4AA;
   // GBK_TO_UNICODE[22861] := 16#83AB;
   // GBK_TO_UNICODE[22862] := 16#C4AB;
   // GBK_TO_UNICODE[22863] := 16#58A8;
   // GBK_TO_UNICODE[22864] := 16#C4AC;
   // GBK_TO_UNICODE[22865] := 16#9ED8;
   // GBK_TO_UNICODE[22866] := 16#C4AD;
   // GBK_TO_UNICODE[22867] := 16#6CAB;
   // GBK_TO_UNICODE[22868] := 16#C4AE;
   // GBK_TO_UNICODE[22869] := 16#6F20;
   // GBK_TO_UNICODE[22870] := 16#C4AF;
   // GBK_TO_UNICODE[22871] := 16#5BDE;
   // GBK_TO_UNICODE[22872] := 16#C4B0;
   // GBK_TO_UNICODE[22873] := 16#964C;
   // GBK_TO_UNICODE[22874] := 16#C4B1;
   // GBK_TO_UNICODE[22875] := 16#8C0B;
   // GBK_TO_UNICODE[22876] := 16#C4B2;
   // GBK_TO_UNICODE[22877] := 16#725F;
   // GBK_TO_UNICODE[22878] := 16#C4B3;
   // GBK_TO_UNICODE[22879] := 16#67D0;
   // GBK_TO_UNICODE[22880] := 16#C4B4;
   // GBK_TO_UNICODE[22881] := 16#62C7;
   // GBK_TO_UNICODE[22882] := 16#C4B5;
   // GBK_TO_UNICODE[22883] := 16#7261;
   // GBK_TO_UNICODE[22884] := 16#C4B6;
   // GBK_TO_UNICODE[22885] := 16#4EA9;
   // GBK_TO_UNICODE[22886] := 16#C4B7;
   // GBK_TO_UNICODE[22887] := 16#59C6;
   // GBK_TO_UNICODE[22888] := 16#C4B8;
   // GBK_TO_UNICODE[22889] := 16#6BCD;
   // GBK_TO_UNICODE[22890] := 16#C4B9;
   // GBK_TO_UNICODE[22891] := 16#5893;
   // GBK_TO_UNICODE[22892] := 16#C4BA;
   // GBK_TO_UNICODE[22893] := 16#66AE;
   // GBK_TO_UNICODE[22894] := 16#C4BB;
   // GBK_TO_UNICODE[22895] := 16#5E55;
   // GBK_TO_UNICODE[22896] := 16#C4BC;
   // GBK_TO_UNICODE[22897] := 16#52DF;
   // GBK_TO_UNICODE[22898] := 16#C4BD;
   // GBK_TO_UNICODE[22899] := 16#6155;
   // GBK_TO_UNICODE[22900] := 16#C4BE;
   // GBK_TO_UNICODE[22901] := 16#6728;
   // GBK_TO_UNICODE[22902] := 16#C4BF;
   // GBK_TO_UNICODE[22903] := 16#76EE;
   // GBK_TO_UNICODE[22904] := 16#C4C0;
   // GBK_TO_UNICODE[22905] := 16#7766;
   // GBK_TO_UNICODE[22906] := 16#C4C1;
   // GBK_TO_UNICODE[22907] := 16#7267;
   // GBK_TO_UNICODE[22908] := 16#C4C2;
   // GBK_TO_UNICODE[22909] := 16#7A46;
   // GBK_TO_UNICODE[22910] := 16#C4C3;
   // GBK_TO_UNICODE[22911] := 16#62FF;
   // GBK_TO_UNICODE[22912] := 16#C4C4;
   // GBK_TO_UNICODE[22913] := 16#54EA;
   // GBK_TO_UNICODE[22914] := 16#C4C5;
   // GBK_TO_UNICODE[22915] := 16#5450;
   // GBK_TO_UNICODE[22916] := 16#C4C6;
   // GBK_TO_UNICODE[22917] := 16#94A0;
   // GBK_TO_UNICODE[22918] := 16#C4C7;
   // GBK_TO_UNICODE[22919] := 16#90A3;
   // GBK_TO_UNICODE[22920] := 16#C4C8;
   // GBK_TO_UNICODE[22921] := 16#5A1C;
   // GBK_TO_UNICODE[22922] := 16#C4C9;
   // GBK_TO_UNICODE[22923] := 16#7EB3;
   // GBK_TO_UNICODE[22924] := 16#C4CA;
   // GBK_TO_UNICODE[22925] := 16#6C16;
   // GBK_TO_UNICODE[22926] := 16#C4CB;
   // GBK_TO_UNICODE[22927] := 16#4E43;
   // GBK_TO_UNICODE[22928] := 16#C4CC;
   // GBK_TO_UNICODE[22929] := 16#5976;
   // GBK_TO_UNICODE[22930] := 16#C4CD;
   // GBK_TO_UNICODE[22931] := 16#8010;
   // GBK_TO_UNICODE[22932] := 16#C4CE;
   // GBK_TO_UNICODE[22933] := 16#5948;
   // GBK_TO_UNICODE[22934] := 16#C4CF;
   // GBK_TO_UNICODE[22935] := 16#5357;
   // GBK_TO_UNICODE[22936] := 16#C4D0;
   // GBK_TO_UNICODE[22937] := 16#7537;
   // GBK_TO_UNICODE[22938] := 16#C4D1;
   // GBK_TO_UNICODE[22939] := 16#96BE;
   // GBK_TO_UNICODE[22940] := 16#C4D2;
   // GBK_TO_UNICODE[22941] := 16#56CA;
   // GBK_TO_UNICODE[22942] := 16#C4D3;
   // GBK_TO_UNICODE[22943] := 16#6320;
   // GBK_TO_UNICODE[22944] := 16#C4D4;
   // GBK_TO_UNICODE[22945] := 16#8111;
   // GBK_TO_UNICODE[22946] := 16#C4D5;
   // GBK_TO_UNICODE[22947] := 16#607C;
   // GBK_TO_UNICODE[22948] := 16#C4D6;
   // GBK_TO_UNICODE[22949] := 16#95F9;
   // GBK_TO_UNICODE[22950] := 16#C4D7;
   // GBK_TO_UNICODE[22951] := 16#6DD6;
   // GBK_TO_UNICODE[22952] := 16#C4D8;
   // GBK_TO_UNICODE[22953] := 16#5462;
   // GBK_TO_UNICODE[22954] := 16#C4D9;
   // GBK_TO_UNICODE[22955] := 16#9981;
   // GBK_TO_UNICODE[22956] := 16#C4DA;
   // GBK_TO_UNICODE[22957] := 16#5185;
   // GBK_TO_UNICODE[22958] := 16#C4DB;
   // GBK_TO_UNICODE[22959] := 16#5AE9;
   // GBK_TO_UNICODE[22960] := 16#C4DC;
   // GBK_TO_UNICODE[22961] := 16#80FD;
   // GBK_TO_UNICODE[22962] := 16#C4DD;
   // GBK_TO_UNICODE[22963] := 16#59AE;
   // GBK_TO_UNICODE[22964] := 16#C4DE;
   // GBK_TO_UNICODE[22965] := 16#9713;
   // GBK_TO_UNICODE[22966] := 16#C4DF;
   // GBK_TO_UNICODE[22967] := 16#502A;
   // GBK_TO_UNICODE[22968] := 16#C4E0;
   // GBK_TO_UNICODE[22969] := 16#6CE5;
   // GBK_TO_UNICODE[22970] := 16#C4E1;
   // GBK_TO_UNICODE[22971] := 16#5C3C;
   // GBK_TO_UNICODE[22972] := 16#C4E2;
   // GBK_TO_UNICODE[22973] := 16#62DF;
   // GBK_TO_UNICODE[22974] := 16#C4E3;
   // GBK_TO_UNICODE[22975] := 16#4F60;
   // GBK_TO_UNICODE[22976] := 16#C4E4;
   // GBK_TO_UNICODE[22977] := 16#533F;
   // GBK_TO_UNICODE[22978] := 16#C4E5;
   // GBK_TO_UNICODE[22979] := 16#817B;
   // GBK_TO_UNICODE[22980] := 16#C4E6;
   // GBK_TO_UNICODE[22981] := 16#9006;
   // GBK_TO_UNICODE[22982] := 16#C4E7;
   // GBK_TO_UNICODE[22983] := 16#6EBA;
   // GBK_TO_UNICODE[22984] := 16#C4E8;
   // GBK_TO_UNICODE[22985] := 16#852B;
   // GBK_TO_UNICODE[22986] := 16#C4E9;
   // GBK_TO_UNICODE[22987] := 16#62C8;
   // GBK_TO_UNICODE[22988] := 16#C4EA;
   // GBK_TO_UNICODE[22989] := 16#5E74;
   // GBK_TO_UNICODE[22990] := 16#C4EB;
   // GBK_TO_UNICODE[22991] := 16#78BE;
   // GBK_TO_UNICODE[22992] := 16#C4EC;
   // GBK_TO_UNICODE[22993] := 16#64B5;
   // GBK_TO_UNICODE[22994] := 16#C4ED;
   // GBK_TO_UNICODE[22995] := 16#637B;
   // GBK_TO_UNICODE[22996] := 16#C4EE;
   // GBK_TO_UNICODE[22997] := 16#5FF5;
   // GBK_TO_UNICODE[22998] := 16#C4EF;
   // GBK_TO_UNICODE[22999] := 16#5A18;
   // GBK_TO_UNICODE[23000] := 16#C4F0;
   // GBK_TO_UNICODE[23001] := 16#917F;
   // GBK_TO_UNICODE[23002] := 16#C4F1;
   // GBK_TO_UNICODE[23003] := 16#9E1F;
   // GBK_TO_UNICODE[23004] := 16#C4F2;
   // GBK_TO_UNICODE[23005] := 16#5C3F;
   // GBK_TO_UNICODE[23006] := 16#C4F3;
   // GBK_TO_UNICODE[23007] := 16#634F;
   // GBK_TO_UNICODE[23008] := 16#C4F4;
   // GBK_TO_UNICODE[23009] := 16#8042;
   // GBK_TO_UNICODE[23010] := 16#C4F5;
   // GBK_TO_UNICODE[23011] := 16#5B7D;
   // GBK_TO_UNICODE[23012] := 16#C4F6;
   // GBK_TO_UNICODE[23013] := 16#556E;
   // GBK_TO_UNICODE[23014] := 16#C4F7;
   // GBK_TO_UNICODE[23015] := 16#954A;
   // GBK_TO_UNICODE[23016] := 16#C4F8;
   // GBK_TO_UNICODE[23017] := 16#954D;
   // GBK_TO_UNICODE[23018] := 16#C4F9;
   // GBK_TO_UNICODE[23019] := 16#6D85;
   // GBK_TO_UNICODE[23020] := 16#C4FA;
   // GBK_TO_UNICODE[23021] := 16#60A8;
   // GBK_TO_UNICODE[23022] := 16#C4FB;
   // GBK_TO_UNICODE[23023] := 16#67E0;
   // GBK_TO_UNICODE[23024] := 16#C4FC;
   // GBK_TO_UNICODE[23025] := 16#72DE;
   // GBK_TO_UNICODE[23026] := 16#C4FD;
   // GBK_TO_UNICODE[23027] := 16#51DD;
   // GBK_TO_UNICODE[23028] := 16#C4FE;
   // GBK_TO_UNICODE[23029] := 16#5B81;
   // GBK_TO_UNICODE[23030] := 16#C540;
   // GBK_TO_UNICODE[23031] := 16#81D4;
   // GBK_TO_UNICODE[23032] := 16#C541;
   // GBK_TO_UNICODE[23033] := 16#81D5;
   // GBK_TO_UNICODE[23034] := 16#C542;
   // GBK_TO_UNICODE[23035] := 16#81D6;
   // GBK_TO_UNICODE[23036] := 16#C543;
   // GBK_TO_UNICODE[23037] := 16#81D7;
   // GBK_TO_UNICODE[23038] := 16#C544;
   // GBK_TO_UNICODE[23039] := 16#81D8;
   // GBK_TO_UNICODE[23040] := 16#C545;
   // GBK_TO_UNICODE[23041] := 16#81D9;
   // GBK_TO_UNICODE[23042] := 16#C546;
   // GBK_TO_UNICODE[23043] := 16#81DA;
   // GBK_TO_UNICODE[23044] := 16#C547;
   // GBK_TO_UNICODE[23045] := 16#81DB;
   // GBK_TO_UNICODE[23046] := 16#C548;
   // GBK_TO_UNICODE[23047] := 16#81DC;
   // GBK_TO_UNICODE[23048] := 16#C549;
   // GBK_TO_UNICODE[23049] := 16#81DD;
   // GBK_TO_UNICODE[23050] := 16#C54A;
   // GBK_TO_UNICODE[23051] := 16#81DE;
   // GBK_TO_UNICODE[23052] := 16#C54B;
   // GBK_TO_UNICODE[23053] := 16#81DF;
   // GBK_TO_UNICODE[23054] := 16#C54C;
   // GBK_TO_UNICODE[23055] := 16#81E0;
   // GBK_TO_UNICODE[23056] := 16#C54D;
   // GBK_TO_UNICODE[23057] := 16#81E1;
   // GBK_TO_UNICODE[23058] := 16#C54E;
   // GBK_TO_UNICODE[23059] := 16#81E2;
   // GBK_TO_UNICODE[23060] := 16#C54F;
   // GBK_TO_UNICODE[23061] := 16#81E4;
   // GBK_TO_UNICODE[23062] := 16#C550;
   // GBK_TO_UNICODE[23063] := 16#81E5;
   // GBK_TO_UNICODE[23064] := 16#C551;
   // GBK_TO_UNICODE[23065] := 16#81E6;
   // GBK_TO_UNICODE[23066] := 16#C552;
   // GBK_TO_UNICODE[23067] := 16#81E8;
   // GBK_TO_UNICODE[23068] := 16#C553;
   // GBK_TO_UNICODE[23069] := 16#81E9;
   // GBK_TO_UNICODE[23070] := 16#C554;
   // GBK_TO_UNICODE[23071] := 16#81EB;
   // GBK_TO_UNICODE[23072] := 16#C555;
   // GBK_TO_UNICODE[23073] := 16#81EE;
   // GBK_TO_UNICODE[23074] := 16#C556;
   // GBK_TO_UNICODE[23075] := 16#81EF;
   // GBK_TO_UNICODE[23076] := 16#C557;
   // GBK_TO_UNICODE[23077] := 16#81F0;
   // GBK_TO_UNICODE[23078] := 16#C558;
   // GBK_TO_UNICODE[23079] := 16#81F1;
   // GBK_TO_UNICODE[23080] := 16#C559;
   // GBK_TO_UNICODE[23081] := 16#81F2;
   // GBK_TO_UNICODE[23082] := 16#C55A;
   // GBK_TO_UNICODE[23083] := 16#81F5;
   // GBK_TO_UNICODE[23084] := 16#C55B;
   // GBK_TO_UNICODE[23085] := 16#81F6;
   // GBK_TO_UNICODE[23086] := 16#C55C;
   // GBK_TO_UNICODE[23087] := 16#81F7;
   // GBK_TO_UNICODE[23088] := 16#C55D;
   // GBK_TO_UNICODE[23089] := 16#81F8;
   // GBK_TO_UNICODE[23090] := 16#C55E;
   // GBK_TO_UNICODE[23091] := 16#81F9;
   // GBK_TO_UNICODE[23092] := 16#C55F;
   // GBK_TO_UNICODE[23093] := 16#81FA;
   // GBK_TO_UNICODE[23094] := 16#C560;
   // GBK_TO_UNICODE[23095] := 16#81FD;
   // GBK_TO_UNICODE[23096] := 16#C561;
   // GBK_TO_UNICODE[23097] := 16#81FF;
   // GBK_TO_UNICODE[23098] := 16#C562;
   // GBK_TO_UNICODE[23099] := 16#8203;
   // GBK_TO_UNICODE[23100] := 16#C563;
   // GBK_TO_UNICODE[23101] := 16#8207;
   // GBK_TO_UNICODE[23102] := 16#C564;
   // GBK_TO_UNICODE[23103] := 16#8208;
   // GBK_TO_UNICODE[23104] := 16#C565;
   // GBK_TO_UNICODE[23105] := 16#8209;
   // GBK_TO_UNICODE[23106] := 16#C566;
   // GBK_TO_UNICODE[23107] := 16#820A;
   // GBK_TO_UNICODE[23108] := 16#C567;
   // GBK_TO_UNICODE[23109] := 16#820B;
   // GBK_TO_UNICODE[23110] := 16#C568;
   // GBK_TO_UNICODE[23111] := 16#820E;
   // GBK_TO_UNICODE[23112] := 16#C569;
   // GBK_TO_UNICODE[23113] := 16#820F;
   // GBK_TO_UNICODE[23114] := 16#C56A;
   // GBK_TO_UNICODE[23115] := 16#8211;
   // GBK_TO_UNICODE[23116] := 16#C56B;
   // GBK_TO_UNICODE[23117] := 16#8213;
   // GBK_TO_UNICODE[23118] := 16#C56C;
   // GBK_TO_UNICODE[23119] := 16#8215;
   // GBK_TO_UNICODE[23120] := 16#C56D;
   // GBK_TO_UNICODE[23121] := 16#8216;
   // GBK_TO_UNICODE[23122] := 16#C56E;
   // GBK_TO_UNICODE[23123] := 16#8217;
   // GBK_TO_UNICODE[23124] := 16#C56F;
   // GBK_TO_UNICODE[23125] := 16#8218;
   // GBK_TO_UNICODE[23126] := 16#C570;
   // GBK_TO_UNICODE[23127] := 16#8219;
   // GBK_TO_UNICODE[23128] := 16#C571;
   // GBK_TO_UNICODE[23129] := 16#821A;
   // GBK_TO_UNICODE[23130] := 16#C572;
   // GBK_TO_UNICODE[23131] := 16#821D;
   // GBK_TO_UNICODE[23132] := 16#C573;
   // GBK_TO_UNICODE[23133] := 16#8220;
   // GBK_TO_UNICODE[23134] := 16#C574;
   // GBK_TO_UNICODE[23135] := 16#8224;
   // GBK_TO_UNICODE[23136] := 16#C575;
   // GBK_TO_UNICODE[23137] := 16#8225;
   // GBK_TO_UNICODE[23138] := 16#C576;
   // GBK_TO_UNICODE[23139] := 16#8226;
   // GBK_TO_UNICODE[23140] := 16#C577;
   // GBK_TO_UNICODE[23141] := 16#8227;
   // GBK_TO_UNICODE[23142] := 16#C578;
   // GBK_TO_UNICODE[23143] := 16#8229;
   // GBK_TO_UNICODE[23144] := 16#C579;
   // GBK_TO_UNICODE[23145] := 16#822E;
   // GBK_TO_UNICODE[23146] := 16#C57A;
   // GBK_TO_UNICODE[23147] := 16#8232;
   // GBK_TO_UNICODE[23148] := 16#C57B;
   // GBK_TO_UNICODE[23149] := 16#823A;
   // GBK_TO_UNICODE[23150] := 16#C57C;
   // GBK_TO_UNICODE[23151] := 16#823C;
   // GBK_TO_UNICODE[23152] := 16#C57D;
   // GBK_TO_UNICODE[23153] := 16#823D;
   // GBK_TO_UNICODE[23154] := 16#C57E;
   // GBK_TO_UNICODE[23155] := 16#823F;
   // GBK_TO_UNICODE[23156] := 16#C580;
   // GBK_TO_UNICODE[23157] := 16#8240;
   // GBK_TO_UNICODE[23158] := 16#C581;
   // GBK_TO_UNICODE[23159] := 16#8241;
   // GBK_TO_UNICODE[23160] := 16#C582;
   // GBK_TO_UNICODE[23161] := 16#8242;
   // GBK_TO_UNICODE[23162] := 16#C583;
   // GBK_TO_UNICODE[23163] := 16#8243;
   // GBK_TO_UNICODE[23164] := 16#C584;
   // GBK_TO_UNICODE[23165] := 16#8245;
   // GBK_TO_UNICODE[23166] := 16#C585;
   // GBK_TO_UNICODE[23167] := 16#8246;
   // GBK_TO_UNICODE[23168] := 16#C586;
   // GBK_TO_UNICODE[23169] := 16#8248;
   // GBK_TO_UNICODE[23170] := 16#C587;
   // GBK_TO_UNICODE[23171] := 16#824A;
   // GBK_TO_UNICODE[23172] := 16#C588;
   // GBK_TO_UNICODE[23173] := 16#824C;
   // GBK_TO_UNICODE[23174] := 16#C589;
   // GBK_TO_UNICODE[23175] := 16#824D;
   // GBK_TO_UNICODE[23176] := 16#C58A;
   // GBK_TO_UNICODE[23177] := 16#824E;
   // GBK_TO_UNICODE[23178] := 16#C58B;
   // GBK_TO_UNICODE[23179] := 16#8250;
   // GBK_TO_UNICODE[23180] := 16#C58C;
   // GBK_TO_UNICODE[23181] := 16#8251;
   // GBK_TO_UNICODE[23182] := 16#C58D;
   // GBK_TO_UNICODE[23183] := 16#8252;
   // GBK_TO_UNICODE[23184] := 16#C58E;
   // GBK_TO_UNICODE[23185] := 16#8253;
   // GBK_TO_UNICODE[23186] := 16#C58F;
   // GBK_TO_UNICODE[23187] := 16#8254;
   // GBK_TO_UNICODE[23188] := 16#C590;
   // GBK_TO_UNICODE[23189] := 16#8255;
   // GBK_TO_UNICODE[23190] := 16#C591;
   // GBK_TO_UNICODE[23191] := 16#8256;
   // GBK_TO_UNICODE[23192] := 16#C592;
   // GBK_TO_UNICODE[23193] := 16#8257;
   // GBK_TO_UNICODE[23194] := 16#C593;
   // GBK_TO_UNICODE[23195] := 16#8259;
   // GBK_TO_UNICODE[23196] := 16#C594;
   // GBK_TO_UNICODE[23197] := 16#825B;
   // GBK_TO_UNICODE[23198] := 16#C595;
   // GBK_TO_UNICODE[23199] := 16#825C;
   // GBK_TO_UNICODE[23200] := 16#C596;
   // GBK_TO_UNICODE[23201] := 16#825D;
   // GBK_TO_UNICODE[23202] := 16#C597;
   // GBK_TO_UNICODE[23203] := 16#825E;
   // GBK_TO_UNICODE[23204] := 16#C598;
   // GBK_TO_UNICODE[23205] := 16#8260;
   // GBK_TO_UNICODE[23206] := 16#C599;
   // GBK_TO_UNICODE[23207] := 16#8261;
   // GBK_TO_UNICODE[23208] := 16#C59A;
   // GBK_TO_UNICODE[23209] := 16#8262;
   // GBK_TO_UNICODE[23210] := 16#C59B;
   // GBK_TO_UNICODE[23211] := 16#8263;
   // GBK_TO_UNICODE[23212] := 16#C59C;
   // GBK_TO_UNICODE[23213] := 16#8264;
   // GBK_TO_UNICODE[23214] := 16#C59D;
   // GBK_TO_UNICODE[23215] := 16#8265;
   // GBK_TO_UNICODE[23216] := 16#C59E;
   // GBK_TO_UNICODE[23217] := 16#8266;
   // GBK_TO_UNICODE[23218] := 16#C59F;
   // GBK_TO_UNICODE[23219] := 16#8267;
   // GBK_TO_UNICODE[23220] := 16#C5A0;
   // GBK_TO_UNICODE[23221] := 16#8269;
   // GBK_TO_UNICODE[23222] := 16#C5A1;
   // GBK_TO_UNICODE[23223] := 16#62E7;
   // GBK_TO_UNICODE[23224] := 16#C5A2;
   // GBK_TO_UNICODE[23225] := 16#6CDE;
   // GBK_TO_UNICODE[23226] := 16#C5A3;
   // GBK_TO_UNICODE[23227] := 16#725B;
   // GBK_TO_UNICODE[23228] := 16#C5A4;
   // GBK_TO_UNICODE[23229] := 16#626D;
   // GBK_TO_UNICODE[23230] := 16#C5A5;
   // GBK_TO_UNICODE[23231] := 16#94AE;
   // GBK_TO_UNICODE[23232] := 16#C5A6;
   // GBK_TO_UNICODE[23233] := 16#7EBD;
   // GBK_TO_UNICODE[23234] := 16#C5A7;
   // GBK_TO_UNICODE[23235] := 16#8113;
   // GBK_TO_UNICODE[23236] := 16#C5A8;
   // GBK_TO_UNICODE[23237] := 16#6D53;
   // GBK_TO_UNICODE[23238] := 16#C5A9;
   // GBK_TO_UNICODE[23239] := 16#519C;
   // GBK_TO_UNICODE[23240] := 16#C5AA;
   // GBK_TO_UNICODE[23241] := 16#5F04;
   // GBK_TO_UNICODE[23242] := 16#C5AB;
   // GBK_TO_UNICODE[23243] := 16#5974;
   // GBK_TO_UNICODE[23244] := 16#C5AC;
   // GBK_TO_UNICODE[23245] := 16#52AA;
   // GBK_TO_UNICODE[23246] := 16#C5AD;
   // GBK_TO_UNICODE[23247] := 16#6012;
   // GBK_TO_UNICODE[23248] := 16#C5AE;
   // GBK_TO_UNICODE[23249] := 16#5973;
   // GBK_TO_UNICODE[23250] := 16#C5AF;
   // GBK_TO_UNICODE[23251] := 16#6696;
   // GBK_TO_UNICODE[23252] := 16#C5B0;
   // GBK_TO_UNICODE[23253] := 16#8650;
   // GBK_TO_UNICODE[23254] := 16#C5B1;
   // GBK_TO_UNICODE[23255] := 16#759F;
   // GBK_TO_UNICODE[23256] := 16#C5B2;
   // GBK_TO_UNICODE[23257] := 16#632A;
   // GBK_TO_UNICODE[23258] := 16#C5B3;
   // GBK_TO_UNICODE[23259] := 16#61E6;
   // GBK_TO_UNICODE[23260] := 16#C5B4;
   // GBK_TO_UNICODE[23261] := 16#7CEF;
   // GBK_TO_UNICODE[23262] := 16#C5B5;
   // GBK_TO_UNICODE[23263] := 16#8BFA;
   // GBK_TO_UNICODE[23264] := 16#C5B6;
   // GBK_TO_UNICODE[23265] := 16#54E6;
   // GBK_TO_UNICODE[23266] := 16#C5B7;
   // GBK_TO_UNICODE[23267] := 16#6B27;
   // GBK_TO_UNICODE[23268] := 16#C5B8;
   // GBK_TO_UNICODE[23269] := 16#9E25;
   // GBK_TO_UNICODE[23270] := 16#C5B9;
   // GBK_TO_UNICODE[23271] := 16#6BB4;
   // GBK_TO_UNICODE[23272] := 16#C5BA;
   // GBK_TO_UNICODE[23273] := 16#85D5;
   // GBK_TO_UNICODE[23274] := 16#C5BB;
   // GBK_TO_UNICODE[23275] := 16#5455;
   // GBK_TO_UNICODE[23276] := 16#C5BC;
   // GBK_TO_UNICODE[23277] := 16#5076;
   // GBK_TO_UNICODE[23278] := 16#C5BD;
   // GBK_TO_UNICODE[23279] := 16#6CA4;
   // GBK_TO_UNICODE[23280] := 16#C5BE;
   // GBK_TO_UNICODE[23281] := 16#556A;
   // GBK_TO_UNICODE[23282] := 16#C5BF;
   // GBK_TO_UNICODE[23283] := 16#8DB4;
   // GBK_TO_UNICODE[23284] := 16#C5C0;
   // GBK_TO_UNICODE[23285] := 16#722C;
   // GBK_TO_UNICODE[23286] := 16#C5C1;
   // GBK_TO_UNICODE[23287] := 16#5E15;
   // GBK_TO_UNICODE[23288] := 16#C5C2;
   // GBK_TO_UNICODE[23289] := 16#6015;
   // GBK_TO_UNICODE[23290] := 16#C5C3;
   // GBK_TO_UNICODE[23291] := 16#7436;
   // GBK_TO_UNICODE[23292] := 16#C5C4;
   // GBK_TO_UNICODE[23293] := 16#62CD;
   // GBK_TO_UNICODE[23294] := 16#C5C5;
   // GBK_TO_UNICODE[23295] := 16#6392;
   // GBK_TO_UNICODE[23296] := 16#C5C6;
   // GBK_TO_UNICODE[23297] := 16#724C;
   // GBK_TO_UNICODE[23298] := 16#C5C7;
   // GBK_TO_UNICODE[23299] := 16#5F98;
   // GBK_TO_UNICODE[23300] := 16#C5C8;
   // GBK_TO_UNICODE[23301] := 16#6E43;
   // GBK_TO_UNICODE[23302] := 16#C5C9;
   // GBK_TO_UNICODE[23303] := 16#6D3E;
   // GBK_TO_UNICODE[23304] := 16#C5CA;
   // GBK_TO_UNICODE[23305] := 16#6500;
   // GBK_TO_UNICODE[23306] := 16#C5CB;
   // GBK_TO_UNICODE[23307] := 16#6F58;
   // GBK_TO_UNICODE[23308] := 16#C5CC;
   // GBK_TO_UNICODE[23309] := 16#76D8;
   // GBK_TO_UNICODE[23310] := 16#C5CD;
   // GBK_TO_UNICODE[23311] := 16#78D0;
   // GBK_TO_UNICODE[23312] := 16#C5CE;
   // GBK_TO_UNICODE[23313] := 16#76FC;
   // GBK_TO_UNICODE[23314] := 16#C5CF;
   // GBK_TO_UNICODE[23315] := 16#7554;
   // GBK_TO_UNICODE[23316] := 16#C5D0;
   // GBK_TO_UNICODE[23317] := 16#5224;
   // GBK_TO_UNICODE[23318] := 16#C5D1;
   // GBK_TO_UNICODE[23319] := 16#53DB;
   // GBK_TO_UNICODE[23320] := 16#C5D2;
   // GBK_TO_UNICODE[23321] := 16#4E53;
   // GBK_TO_UNICODE[23322] := 16#C5D3;
   // GBK_TO_UNICODE[23323] := 16#5E9E;
   // GBK_TO_UNICODE[23324] := 16#C5D4;
   // GBK_TO_UNICODE[23325] := 16#65C1;
   // GBK_TO_UNICODE[23326] := 16#C5D5;
   // GBK_TO_UNICODE[23327] := 16#802A;
   // GBK_TO_UNICODE[23328] := 16#C5D6;
   // GBK_TO_UNICODE[23329] := 16#80D6;
   // GBK_TO_UNICODE[23330] := 16#C5D7;
   // GBK_TO_UNICODE[23331] := 16#629B;
   // GBK_TO_UNICODE[23332] := 16#C5D8;
   // GBK_TO_UNICODE[23333] := 16#5486;
   // GBK_TO_UNICODE[23334] := 16#C5D9;
   // GBK_TO_UNICODE[23335] := 16#5228;
   // GBK_TO_UNICODE[23336] := 16#C5DA;
   // GBK_TO_UNICODE[23337] := 16#70AE;
   // GBK_TO_UNICODE[23338] := 16#C5DB;
   // GBK_TO_UNICODE[23339] := 16#888D;
   // GBK_TO_UNICODE[23340] := 16#C5DC;
   // GBK_TO_UNICODE[23341] := 16#8DD1;
   // GBK_TO_UNICODE[23342] := 16#C5DD;
   // GBK_TO_UNICODE[23343] := 16#6CE1;
   // GBK_TO_UNICODE[23344] := 16#C5DE;
   // GBK_TO_UNICODE[23345] := 16#5478;
   // GBK_TO_UNICODE[23346] := 16#C5DF;
   // GBK_TO_UNICODE[23347] := 16#80DA;
   // GBK_TO_UNICODE[23348] := 16#C5E0;
   // GBK_TO_UNICODE[23349] := 16#57F9;
   // GBK_TO_UNICODE[23350] := 16#C5E1;
   // GBK_TO_UNICODE[23351] := 16#88F4;
   // GBK_TO_UNICODE[23352] := 16#C5E2;
   // GBK_TO_UNICODE[23353] := 16#8D54;
   // GBK_TO_UNICODE[23354] := 16#C5E3;
   // GBK_TO_UNICODE[23355] := 16#966A;
   // GBK_TO_UNICODE[23356] := 16#C5E4;
   // GBK_TO_UNICODE[23357] := 16#914D;
   // GBK_TO_UNICODE[23358] := 16#C5E5;
   // GBK_TO_UNICODE[23359] := 16#4F69;
   // GBK_TO_UNICODE[23360] := 16#C5E6;
   // GBK_TO_UNICODE[23361] := 16#6C9B;
   // GBK_TO_UNICODE[23362] := 16#C5E7;
   // GBK_TO_UNICODE[23363] := 16#55B7;
   // GBK_TO_UNICODE[23364] := 16#C5E8;
   // GBK_TO_UNICODE[23365] := 16#76C6;
   // GBK_TO_UNICODE[23366] := 16#C5E9;
   // GBK_TO_UNICODE[23367] := 16#7830;
   // GBK_TO_UNICODE[23368] := 16#C5EA;
   // GBK_TO_UNICODE[23369] := 16#62A8;
   // GBK_TO_UNICODE[23370] := 16#C5EB;
   // GBK_TO_UNICODE[23371] := 16#70F9;
   // GBK_TO_UNICODE[23372] := 16#C5EC;
   // GBK_TO_UNICODE[23373] := 16#6F8E;
   // GBK_TO_UNICODE[23374] := 16#C5ED;
   // GBK_TO_UNICODE[23375] := 16#5F6D;
   // GBK_TO_UNICODE[23376] := 16#C5EE;
   // GBK_TO_UNICODE[23377] := 16#84EC;
   // GBK_TO_UNICODE[23378] := 16#C5EF;
   // GBK_TO_UNICODE[23379] := 16#68DA;
   // GBK_TO_UNICODE[23380] := 16#C5F0;
   // GBK_TO_UNICODE[23381] := 16#787C;
   // GBK_TO_UNICODE[23382] := 16#C5F1;
   // GBK_TO_UNICODE[23383] := 16#7BF7;
   // GBK_TO_UNICODE[23384] := 16#C5F2;
   // GBK_TO_UNICODE[23385] := 16#81A8;
   // GBK_TO_UNICODE[23386] := 16#C5F3;
   // GBK_TO_UNICODE[23387] := 16#670B;
   // GBK_TO_UNICODE[23388] := 16#C5F4;
   // GBK_TO_UNICODE[23389] := 16#9E4F;
   // GBK_TO_UNICODE[23390] := 16#C5F5;
   // GBK_TO_UNICODE[23391] := 16#6367;
   // GBK_TO_UNICODE[23392] := 16#C5F6;
   // GBK_TO_UNICODE[23393] := 16#78B0;
   // GBK_TO_UNICODE[23394] := 16#C5F7;
   // GBK_TO_UNICODE[23395] := 16#576F;
   // GBK_TO_UNICODE[23396] := 16#C5F8;
   // GBK_TO_UNICODE[23397] := 16#7812;
   // GBK_TO_UNICODE[23398] := 16#C5F9;
   // GBK_TO_UNICODE[23399] := 16#9739;
   // GBK_TO_UNICODE[23400] := 16#C5FA;
   // GBK_TO_UNICODE[23401] := 16#6279;
   // GBK_TO_UNICODE[23402] := 16#C5FB;
   // GBK_TO_UNICODE[23403] := 16#62AB;
   // GBK_TO_UNICODE[23404] := 16#C5FC;
   // GBK_TO_UNICODE[23405] := 16#5288;
   // GBK_TO_UNICODE[23406] := 16#C5FD;
   // GBK_TO_UNICODE[23407] := 16#7435;
   // GBK_TO_UNICODE[23408] := 16#C5FE;
   // GBK_TO_UNICODE[23409] := 16#6BD7;
   // GBK_TO_UNICODE[23410] := 16#C640;
   // GBK_TO_UNICODE[23411] := 16#826A;
   // GBK_TO_UNICODE[23412] := 16#C641;
   // GBK_TO_UNICODE[23413] := 16#826B;
   // GBK_TO_UNICODE[23414] := 16#C642;
   // GBK_TO_UNICODE[23415] := 16#826C;
   // GBK_TO_UNICODE[23416] := 16#C643;
   // GBK_TO_UNICODE[23417] := 16#826D;
   // GBK_TO_UNICODE[23418] := 16#C644;
   // GBK_TO_UNICODE[23419] := 16#8271;
   // GBK_TO_UNICODE[23420] := 16#C645;
   // GBK_TO_UNICODE[23421] := 16#8275;
   // GBK_TO_UNICODE[23422] := 16#C646;
   // GBK_TO_UNICODE[23423] := 16#8276;
   // GBK_TO_UNICODE[23424] := 16#C647;
   // GBK_TO_UNICODE[23425] := 16#8277;
   // GBK_TO_UNICODE[23426] := 16#C648;
   // GBK_TO_UNICODE[23427] := 16#8278;
   // GBK_TO_UNICODE[23428] := 16#C649;
   // GBK_TO_UNICODE[23429] := 16#827B;
   // GBK_TO_UNICODE[23430] := 16#C64A;
   // GBK_TO_UNICODE[23431] := 16#827C;
   // GBK_TO_UNICODE[23432] := 16#C64B;
   // GBK_TO_UNICODE[23433] := 16#8280;
   // GBK_TO_UNICODE[23434] := 16#C64C;
   // GBK_TO_UNICODE[23435] := 16#8281;
   // GBK_TO_UNICODE[23436] := 16#C64D;
   // GBK_TO_UNICODE[23437] := 16#8283;
   // GBK_TO_UNICODE[23438] := 16#C64E;
   // GBK_TO_UNICODE[23439] := 16#8285;
   // GBK_TO_UNICODE[23440] := 16#C64F;
   // GBK_TO_UNICODE[23441] := 16#8286;
   // GBK_TO_UNICODE[23442] := 16#C650;
   // GBK_TO_UNICODE[23443] := 16#8287;
   // GBK_TO_UNICODE[23444] := 16#C651;
   // GBK_TO_UNICODE[23445] := 16#8289;
   // GBK_TO_UNICODE[23446] := 16#C652;
   // GBK_TO_UNICODE[23447] := 16#828C;
   // GBK_TO_UNICODE[23448] := 16#C653;
   // GBK_TO_UNICODE[23449] := 16#8290;
   // GBK_TO_UNICODE[23450] := 16#C654;
   // GBK_TO_UNICODE[23451] := 16#8293;
   // GBK_TO_UNICODE[23452] := 16#C655;
   // GBK_TO_UNICODE[23453] := 16#8294;
   // GBK_TO_UNICODE[23454] := 16#C656;
   // GBK_TO_UNICODE[23455] := 16#8295;
   // GBK_TO_UNICODE[23456] := 16#C657;
   // GBK_TO_UNICODE[23457] := 16#8296;
   // GBK_TO_UNICODE[23458] := 16#C658;
   // GBK_TO_UNICODE[23459] := 16#829A;
   // GBK_TO_UNICODE[23460] := 16#C659;
   // GBK_TO_UNICODE[23461] := 16#829B;
   // GBK_TO_UNICODE[23462] := 16#C65A;
   // GBK_TO_UNICODE[23463] := 16#829E;
   // GBK_TO_UNICODE[23464] := 16#C65B;
   // GBK_TO_UNICODE[23465] := 16#82A0;
   // GBK_TO_UNICODE[23466] := 16#C65C;
   // GBK_TO_UNICODE[23467] := 16#82A2;
   // GBK_TO_UNICODE[23468] := 16#C65D;
   // GBK_TO_UNICODE[23469] := 16#82A3;
   // GBK_TO_UNICODE[23470] := 16#C65E;
   // GBK_TO_UNICODE[23471] := 16#82A7;
   // GBK_TO_UNICODE[23472] := 16#C65F;
   // GBK_TO_UNICODE[23473] := 16#82B2;
   // GBK_TO_UNICODE[23474] := 16#C660;
   // GBK_TO_UNICODE[23475] := 16#82B5;
   // GBK_TO_UNICODE[23476] := 16#C661;
   // GBK_TO_UNICODE[23477] := 16#82B6;
   // GBK_TO_UNICODE[23478] := 16#C662;
   // GBK_TO_UNICODE[23479] := 16#82BA;
   // GBK_TO_UNICODE[23480] := 16#C663;
   // GBK_TO_UNICODE[23481] := 16#82BB;
   // GBK_TO_UNICODE[23482] := 16#C664;
   // GBK_TO_UNICODE[23483] := 16#82BC;
   // GBK_TO_UNICODE[23484] := 16#C665;
   // GBK_TO_UNICODE[23485] := 16#82BF;
   // GBK_TO_UNICODE[23486] := 16#C666;
   // GBK_TO_UNICODE[23487] := 16#82C0;
   // GBK_TO_UNICODE[23488] := 16#C667;
   // GBK_TO_UNICODE[23489] := 16#82C2;
   // GBK_TO_UNICODE[23490] := 16#C668;
   // GBK_TO_UNICODE[23491] := 16#82C3;
   // GBK_TO_UNICODE[23492] := 16#C669;
   // GBK_TO_UNICODE[23493] := 16#82C5;
   // GBK_TO_UNICODE[23494] := 16#C66A;
   // GBK_TO_UNICODE[23495] := 16#82C6;
   // GBK_TO_UNICODE[23496] := 16#C66B;
   // GBK_TO_UNICODE[23497] := 16#82C9;
   // GBK_TO_UNICODE[23498] := 16#C66C;
   // GBK_TO_UNICODE[23499] := 16#82D0;
   // GBK_TO_UNICODE[23500] := 16#C66D;
   // GBK_TO_UNICODE[23501] := 16#82D6;
   // GBK_TO_UNICODE[23502] := 16#C66E;
   // GBK_TO_UNICODE[23503] := 16#82D9;
   // GBK_TO_UNICODE[23504] := 16#C66F;
   // GBK_TO_UNICODE[23505] := 16#82DA;
   // GBK_TO_UNICODE[23506] := 16#C670;
   // GBK_TO_UNICODE[23507] := 16#82DD;
   // GBK_TO_UNICODE[23508] := 16#C671;
   // GBK_TO_UNICODE[23509] := 16#82E2;
   // GBK_TO_UNICODE[23510] := 16#C672;
   // GBK_TO_UNICODE[23511] := 16#82E7;
   // GBK_TO_UNICODE[23512] := 16#C673;
   // GBK_TO_UNICODE[23513] := 16#82E8;
   // GBK_TO_UNICODE[23514] := 16#C674;
   // GBK_TO_UNICODE[23515] := 16#82E9;
   // GBK_TO_UNICODE[23516] := 16#C675;
   // GBK_TO_UNICODE[23517] := 16#82EA;
   // GBK_TO_UNICODE[23518] := 16#C676;
   // GBK_TO_UNICODE[23519] := 16#82EC;
   // GBK_TO_UNICODE[23520] := 16#C677;
   // GBK_TO_UNICODE[23521] := 16#82ED;
   // GBK_TO_UNICODE[23522] := 16#C678;
   // GBK_TO_UNICODE[23523] := 16#82EE;
   // GBK_TO_UNICODE[23524] := 16#C679;
   // GBK_TO_UNICODE[23525] := 16#82F0;
   // GBK_TO_UNICODE[23526] := 16#C67A;
   // GBK_TO_UNICODE[23527] := 16#82F2;
   // GBK_TO_UNICODE[23528] := 16#C67B;
   // GBK_TO_UNICODE[23529] := 16#82F3;
   // GBK_TO_UNICODE[23530] := 16#C67C;
   // GBK_TO_UNICODE[23531] := 16#82F5;
   // GBK_TO_UNICODE[23532] := 16#C67D;
   // GBK_TO_UNICODE[23533] := 16#82F6;
   // GBK_TO_UNICODE[23534] := 16#C67E;
   // GBK_TO_UNICODE[23535] := 16#82F8;
   // GBK_TO_UNICODE[23536] := 16#C680;
   // GBK_TO_UNICODE[23537] := 16#82FA;
   // GBK_TO_UNICODE[23538] := 16#C681;
   // GBK_TO_UNICODE[23539] := 16#82FC;
   // GBK_TO_UNICODE[23540] := 16#C682;
   // GBK_TO_UNICODE[23541] := 16#82FD;
   // GBK_TO_UNICODE[23542] := 16#C683;
   // GBK_TO_UNICODE[23543] := 16#82FE;
   // GBK_TO_UNICODE[23544] := 16#C684;
   // GBK_TO_UNICODE[23545] := 16#82FF;
   // GBK_TO_UNICODE[23546] := 16#C685;
   // GBK_TO_UNICODE[23547] := 16#8300;
   // GBK_TO_UNICODE[23548] := 16#C686;
   // GBK_TO_UNICODE[23549] := 16#830A;
   // GBK_TO_UNICODE[23550] := 16#C687;
   // GBK_TO_UNICODE[23551] := 16#830B;
   // GBK_TO_UNICODE[23552] := 16#C688;
   // GBK_TO_UNICODE[23553] := 16#830D;
   // GBK_TO_UNICODE[23554] := 16#C689;
   // GBK_TO_UNICODE[23555] := 16#8310;
   // GBK_TO_UNICODE[23556] := 16#C68A;
   // GBK_TO_UNICODE[23557] := 16#8312;
   // GBK_TO_UNICODE[23558] := 16#C68B;
   // GBK_TO_UNICODE[23559] := 16#8313;
   // GBK_TO_UNICODE[23560] := 16#C68C;
   // GBK_TO_UNICODE[23561] := 16#8316;
   // GBK_TO_UNICODE[23562] := 16#C68D;
   // GBK_TO_UNICODE[23563] := 16#8318;
   // GBK_TO_UNICODE[23564] := 16#C68E;
   // GBK_TO_UNICODE[23565] := 16#8319;
   // GBK_TO_UNICODE[23566] := 16#C68F;
   // GBK_TO_UNICODE[23567] := 16#831D;
   // GBK_TO_UNICODE[23568] := 16#C690;
   // GBK_TO_UNICODE[23569] := 16#831E;
   // GBK_TO_UNICODE[23570] := 16#C691;
   // GBK_TO_UNICODE[23571] := 16#831F;
   // GBK_TO_UNICODE[23572] := 16#C692;
   // GBK_TO_UNICODE[23573] := 16#8320;
   // GBK_TO_UNICODE[23574] := 16#C693;
   // GBK_TO_UNICODE[23575] := 16#8321;
   // GBK_TO_UNICODE[23576] := 16#C694;
   // GBK_TO_UNICODE[23577] := 16#8322;
   // GBK_TO_UNICODE[23578] := 16#C695;
   // GBK_TO_UNICODE[23579] := 16#8323;
   // GBK_TO_UNICODE[23580] := 16#C696;
   // GBK_TO_UNICODE[23581] := 16#8324;
   // GBK_TO_UNICODE[23582] := 16#C697;
   // GBK_TO_UNICODE[23583] := 16#8325;
   // GBK_TO_UNICODE[23584] := 16#C698;
   // GBK_TO_UNICODE[23585] := 16#8326;
   // GBK_TO_UNICODE[23586] := 16#C699;
   // GBK_TO_UNICODE[23587] := 16#8329;
   // GBK_TO_UNICODE[23588] := 16#C69A;
   // GBK_TO_UNICODE[23589] := 16#832A;
   // GBK_TO_UNICODE[23590] := 16#C69B;
   // GBK_TO_UNICODE[23591] := 16#832E;
   // GBK_TO_UNICODE[23592] := 16#C69C;
   // GBK_TO_UNICODE[23593] := 16#8330;
   // GBK_TO_UNICODE[23594] := 16#C69D;
   // GBK_TO_UNICODE[23595] := 16#8332;
   // GBK_TO_UNICODE[23596] := 16#C69E;
   // GBK_TO_UNICODE[23597] := 16#8337;
   // GBK_TO_UNICODE[23598] := 16#C69F;
   // GBK_TO_UNICODE[23599] := 16#833B;
   // GBK_TO_UNICODE[23600] := 16#C6A0;
   // GBK_TO_UNICODE[23601] := 16#833D;
   // GBK_TO_UNICODE[23602] := 16#C6A1;
   // GBK_TO_UNICODE[23603] := 16#5564;
   // GBK_TO_UNICODE[23604] := 16#C6A2;
   // GBK_TO_UNICODE[23605] := 16#813E;
   // GBK_TO_UNICODE[23606] := 16#C6A3;
   // GBK_TO_UNICODE[23607] := 16#75B2;
   // GBK_TO_UNICODE[23608] := 16#C6A4;
   // GBK_TO_UNICODE[23609] := 16#76AE;
   // GBK_TO_UNICODE[23610] := 16#C6A5;
   // GBK_TO_UNICODE[23611] := 16#5339;
   // GBK_TO_UNICODE[23612] := 16#C6A6;
   // GBK_TO_UNICODE[23613] := 16#75DE;
   // GBK_TO_UNICODE[23614] := 16#C6A7;
   // GBK_TO_UNICODE[23615] := 16#50FB;
   // GBK_TO_UNICODE[23616] := 16#C6A8;
   // GBK_TO_UNICODE[23617] := 16#5C41;
   // GBK_TO_UNICODE[23618] := 16#C6A9;
   // GBK_TO_UNICODE[23619] := 16#8B6C;
   // GBK_TO_UNICODE[23620] := 16#C6AA;
   // GBK_TO_UNICODE[23621] := 16#7BC7;
   // GBK_TO_UNICODE[23622] := 16#C6AB;
   // GBK_TO_UNICODE[23623] := 16#504F;
   // GBK_TO_UNICODE[23624] := 16#C6AC;
   // GBK_TO_UNICODE[23625] := 16#7247;
   // GBK_TO_UNICODE[23626] := 16#C6AD;
   // GBK_TO_UNICODE[23627] := 16#9A97;
   // GBK_TO_UNICODE[23628] := 16#C6AE;
   // GBK_TO_UNICODE[23629] := 16#98D8;
   // GBK_TO_UNICODE[23630] := 16#C6AF;
   // GBK_TO_UNICODE[23631] := 16#6F02;
   // GBK_TO_UNICODE[23632] := 16#C6B0;
   // GBK_TO_UNICODE[23633] := 16#74E2;
   // GBK_TO_UNICODE[23634] := 16#C6B1;
   // GBK_TO_UNICODE[23635] := 16#7968;
   // GBK_TO_UNICODE[23636] := 16#C6B2;
   // GBK_TO_UNICODE[23637] := 16#6487;
   // GBK_TO_UNICODE[23638] := 16#C6B3;
   // GBK_TO_UNICODE[23639] := 16#77A5;
   // GBK_TO_UNICODE[23640] := 16#C6B4;
   // GBK_TO_UNICODE[23641] := 16#62FC;
   // GBK_TO_UNICODE[23642] := 16#C6B5;
   // GBK_TO_UNICODE[23643] := 16#9891;
   // GBK_TO_UNICODE[23644] := 16#C6B6;
   // GBK_TO_UNICODE[23645] := 16#8D2B;
   // GBK_TO_UNICODE[23646] := 16#C6B7;
   // GBK_TO_UNICODE[23647] := 16#54C1;
   // GBK_TO_UNICODE[23648] := 16#C6B8;
   // GBK_TO_UNICODE[23649] := 16#8058;
   // GBK_TO_UNICODE[23650] := 16#C6B9;
   // GBK_TO_UNICODE[23651] := 16#4E52;
   // GBK_TO_UNICODE[23652] := 16#C6BA;
   // GBK_TO_UNICODE[23653] := 16#576A;
   // GBK_TO_UNICODE[23654] := 16#C6BB;
   // GBK_TO_UNICODE[23655] := 16#82F9;
   // GBK_TO_UNICODE[23656] := 16#C6BC;
   // GBK_TO_UNICODE[23657] := 16#840D;
   // GBK_TO_UNICODE[23658] := 16#C6BD;
   // GBK_TO_UNICODE[23659] := 16#5E73;
   // GBK_TO_UNICODE[23660] := 16#C6BE;
   // GBK_TO_UNICODE[23661] := 16#51ED;
   // GBK_TO_UNICODE[23662] := 16#C6BF;
   // GBK_TO_UNICODE[23663] := 16#74F6;
   // GBK_TO_UNICODE[23664] := 16#C6C0;
   // GBK_TO_UNICODE[23665] := 16#8BC4;
   // GBK_TO_UNICODE[23666] := 16#C6C1;
   // GBK_TO_UNICODE[23667] := 16#5C4F;
   // GBK_TO_UNICODE[23668] := 16#C6C2;
   // GBK_TO_UNICODE[23669] := 16#5761;
   // GBK_TO_UNICODE[23670] := 16#C6C3;
   // GBK_TO_UNICODE[23671] := 16#6CFC;
   // GBK_TO_UNICODE[23672] := 16#C6C4;
   // GBK_TO_UNICODE[23673] := 16#9887;
   // GBK_TO_UNICODE[23674] := 16#C6C5;
   // GBK_TO_UNICODE[23675] := 16#5A46;
   // GBK_TO_UNICODE[23676] := 16#C6C6;
   // GBK_TO_UNICODE[23677] := 16#7834;
   // GBK_TO_UNICODE[23678] := 16#C6C7;
   // GBK_TO_UNICODE[23679] := 16#9B44;
   // GBK_TO_UNICODE[23680] := 16#C6C8;
   // GBK_TO_UNICODE[23681] := 16#8FEB;
   // GBK_TO_UNICODE[23682] := 16#C6C9;
   // GBK_TO_UNICODE[23683] := 16#7C95;
   // GBK_TO_UNICODE[23684] := 16#C6CA;
   // GBK_TO_UNICODE[23685] := 16#5256;
   // GBK_TO_UNICODE[23686] := 16#C6CB;
   // GBK_TO_UNICODE[23687] := 16#6251;
   // GBK_TO_UNICODE[23688] := 16#C6CC;
   // GBK_TO_UNICODE[23689] := 16#94FA;
   // GBK_TO_UNICODE[23690] := 16#C6CD;
   // GBK_TO_UNICODE[23691] := 16#4EC6;
   // GBK_TO_UNICODE[23692] := 16#C6CE;
   // GBK_TO_UNICODE[23693] := 16#8386;
   // GBK_TO_UNICODE[23694] := 16#C6CF;
   // GBK_TO_UNICODE[23695] := 16#8461;
   // GBK_TO_UNICODE[23696] := 16#C6D0;
   // GBK_TO_UNICODE[23697] := 16#83E9;
   // GBK_TO_UNICODE[23698] := 16#C6D1;
   // GBK_TO_UNICODE[23699] := 16#84B2;
   // GBK_TO_UNICODE[23700] := 16#C6D2;
   // GBK_TO_UNICODE[23701] := 16#57D4;
   // GBK_TO_UNICODE[23702] := 16#C6D3;
   // GBK_TO_UNICODE[23703] := 16#6734;
   // GBK_TO_UNICODE[23704] := 16#C6D4;
   // GBK_TO_UNICODE[23705] := 16#5703;
   // GBK_TO_UNICODE[23706] := 16#C6D5;
   // GBK_TO_UNICODE[23707] := 16#666E;
   // GBK_TO_UNICODE[23708] := 16#C6D6;
   // GBK_TO_UNICODE[23709] := 16#6D66;
   // GBK_TO_UNICODE[23710] := 16#C6D7;
   // GBK_TO_UNICODE[23711] := 16#8C31;
   // GBK_TO_UNICODE[23712] := 16#C6D8;
   // GBK_TO_UNICODE[23713] := 16#66DD;
   // GBK_TO_UNICODE[23714] := 16#C6D9;
   // GBK_TO_UNICODE[23715] := 16#7011;
   // GBK_TO_UNICODE[23716] := 16#C6DA;
   // GBK_TO_UNICODE[23717] := 16#671F;
   // GBK_TO_UNICODE[23718] := 16#C6DB;
   // GBK_TO_UNICODE[23719] := 16#6B3A;
   // GBK_TO_UNICODE[23720] := 16#C6DC;
   // GBK_TO_UNICODE[23721] := 16#6816;
   // GBK_TO_UNICODE[23722] := 16#C6DD;
   // GBK_TO_UNICODE[23723] := 16#621A;
   // GBK_TO_UNICODE[23724] := 16#C6DE;
   // GBK_TO_UNICODE[23725] := 16#59BB;
   // GBK_TO_UNICODE[23726] := 16#C6DF;
   // GBK_TO_UNICODE[23727] := 16#4E03;
   // GBK_TO_UNICODE[23728] := 16#C6E0;
   // GBK_TO_UNICODE[23729] := 16#51C4;
   // GBK_TO_UNICODE[23730] := 16#C6E1;
   // GBK_TO_UNICODE[23731] := 16#6F06;
   // GBK_TO_UNICODE[23732] := 16#C6E2;
   // GBK_TO_UNICODE[23733] := 16#67D2;
   // GBK_TO_UNICODE[23734] := 16#C6E3;
   // GBK_TO_UNICODE[23735] := 16#6C8F;
   // GBK_TO_UNICODE[23736] := 16#C6E4;
   // GBK_TO_UNICODE[23737] := 16#5176;
   // GBK_TO_UNICODE[23738] := 16#C6E5;
   // GBK_TO_UNICODE[23739] := 16#68CB;
   // GBK_TO_UNICODE[23740] := 16#C6E6;
   // GBK_TO_UNICODE[23741] := 16#5947;
   // GBK_TO_UNICODE[23742] := 16#C6E7;
   // GBK_TO_UNICODE[23743] := 16#6B67;
   // GBK_TO_UNICODE[23744] := 16#C6E8;
   // GBK_TO_UNICODE[23745] := 16#7566;
   // GBK_TO_UNICODE[23746] := 16#C6E9;
   // GBK_TO_UNICODE[23747] := 16#5D0E;
   // GBK_TO_UNICODE[23748] := 16#C6EA;
   // GBK_TO_UNICODE[23749] := 16#8110;
   // GBK_TO_UNICODE[23750] := 16#C6EB;
   // GBK_TO_UNICODE[23751] := 16#9F50;
   // GBK_TO_UNICODE[23752] := 16#C6EC;
   // GBK_TO_UNICODE[23753] := 16#65D7;
   // GBK_TO_UNICODE[23754] := 16#C6ED;
   // GBK_TO_UNICODE[23755] := 16#7948;
   // GBK_TO_UNICODE[23756] := 16#C6EE;
   // GBK_TO_UNICODE[23757] := 16#7941;
   // GBK_TO_UNICODE[23758] := 16#C6EF;
   // GBK_TO_UNICODE[23759] := 16#9A91;
   // GBK_TO_UNICODE[23760] := 16#C6F0;
   // GBK_TO_UNICODE[23761] := 16#8D77;
   // GBK_TO_UNICODE[23762] := 16#C6F1;
   // GBK_TO_UNICODE[23763] := 16#5C82;
   // GBK_TO_UNICODE[23764] := 16#C6F2;
   // GBK_TO_UNICODE[23765] := 16#4E5E;
   // GBK_TO_UNICODE[23766] := 16#C6F3;
   // GBK_TO_UNICODE[23767] := 16#4F01;
   // GBK_TO_UNICODE[23768] := 16#C6F4;
   // GBK_TO_UNICODE[23769] := 16#542F;
   // GBK_TO_UNICODE[23770] := 16#C6F5;
   // GBK_TO_UNICODE[23771] := 16#5951;
   // GBK_TO_UNICODE[23772] := 16#C6F6;
   // GBK_TO_UNICODE[23773] := 16#780C;
   // GBK_TO_UNICODE[23774] := 16#C6F7;
   // GBK_TO_UNICODE[23775] := 16#5668;
   // GBK_TO_UNICODE[23776] := 16#C6F8;
   // GBK_TO_UNICODE[23777] := 16#6C14;
   // GBK_TO_UNICODE[23778] := 16#C6F9;
   // GBK_TO_UNICODE[23779] := 16#8FC4;
   // GBK_TO_UNICODE[23780] := 16#C6FA;
   // GBK_TO_UNICODE[23781] := 16#5F03;
   // GBK_TO_UNICODE[23782] := 16#C6FB;
   // GBK_TO_UNICODE[23783] := 16#6C7D;
   // GBK_TO_UNICODE[23784] := 16#C6FC;
   // GBK_TO_UNICODE[23785] := 16#6CE3;
   // GBK_TO_UNICODE[23786] := 16#C6FD;
   // GBK_TO_UNICODE[23787] := 16#8BAB;
   // GBK_TO_UNICODE[23788] := 16#C6FE;
   // GBK_TO_UNICODE[23789] := 16#6390;
   // GBK_TO_UNICODE[23790] := 16#C740;
   // GBK_TO_UNICODE[23791] := 16#833E;
   // GBK_TO_UNICODE[23792] := 16#C741;
   // GBK_TO_UNICODE[23793] := 16#833F;
   // GBK_TO_UNICODE[23794] := 16#C742;
   // GBK_TO_UNICODE[23795] := 16#8341;
   // GBK_TO_UNICODE[23796] := 16#C743;
   // GBK_TO_UNICODE[23797] := 16#8342;
   // GBK_TO_UNICODE[23798] := 16#C744;
   // GBK_TO_UNICODE[23799] := 16#8344;
   // GBK_TO_UNICODE[23800] := 16#C745;
   // GBK_TO_UNICODE[23801] := 16#8345;
   // GBK_TO_UNICODE[23802] := 16#C746;
   // GBK_TO_UNICODE[23803] := 16#8348;
   // GBK_TO_UNICODE[23804] := 16#C747;
   // GBK_TO_UNICODE[23805] := 16#834A;
   // GBK_TO_UNICODE[23806] := 16#C748;
   // GBK_TO_UNICODE[23807] := 16#834B;
   // GBK_TO_UNICODE[23808] := 16#C749;
   // GBK_TO_UNICODE[23809] := 16#834C;
   // GBK_TO_UNICODE[23810] := 16#C74A;
   // GBK_TO_UNICODE[23811] := 16#834D;
   // GBK_TO_UNICODE[23812] := 16#C74B;
   // GBK_TO_UNICODE[23813] := 16#834E;
   // GBK_TO_UNICODE[23814] := 16#C74C;
   // GBK_TO_UNICODE[23815] := 16#8353;
   // GBK_TO_UNICODE[23816] := 16#C74D;
   // GBK_TO_UNICODE[23817] := 16#8355;
   // GBK_TO_UNICODE[23818] := 16#C74E;
   // GBK_TO_UNICODE[23819] := 16#8356;
   // GBK_TO_UNICODE[23820] := 16#C74F;
   // GBK_TO_UNICODE[23821] := 16#8357;
   // GBK_TO_UNICODE[23822] := 16#C750;
   // GBK_TO_UNICODE[23823] := 16#8358;
   // GBK_TO_UNICODE[23824] := 16#C751;
   // GBK_TO_UNICODE[23825] := 16#8359;
   // GBK_TO_UNICODE[23826] := 16#C752;
   // GBK_TO_UNICODE[23827] := 16#835D;
   // GBK_TO_UNICODE[23828] := 16#C753;
   // GBK_TO_UNICODE[23829] := 16#8362;
   // GBK_TO_UNICODE[23830] := 16#C754;
   // GBK_TO_UNICODE[23831] := 16#8370;
   // GBK_TO_UNICODE[23832] := 16#C755;
   // GBK_TO_UNICODE[23833] := 16#8371;
   // GBK_TO_UNICODE[23834] := 16#C756;
   // GBK_TO_UNICODE[23835] := 16#8372;
   // GBK_TO_UNICODE[23836] := 16#C757;
   // GBK_TO_UNICODE[23837] := 16#8373;
   // GBK_TO_UNICODE[23838] := 16#C758;
   // GBK_TO_UNICODE[23839] := 16#8374;
   // GBK_TO_UNICODE[23840] := 16#C759;
   // GBK_TO_UNICODE[23841] := 16#8375;
   // GBK_TO_UNICODE[23842] := 16#C75A;
   // GBK_TO_UNICODE[23843] := 16#8376;
   // GBK_TO_UNICODE[23844] := 16#C75B;
   // GBK_TO_UNICODE[23845] := 16#8379;
   // GBK_TO_UNICODE[23846] := 16#C75C;
   // GBK_TO_UNICODE[23847] := 16#837A;
   // GBK_TO_UNICODE[23848] := 16#C75D;
   // GBK_TO_UNICODE[23849] := 16#837E;
   // GBK_TO_UNICODE[23850] := 16#C75E;
   // GBK_TO_UNICODE[23851] := 16#837F;
   // GBK_TO_UNICODE[23852] := 16#C75F;
   // GBK_TO_UNICODE[23853] := 16#8380;
   // GBK_TO_UNICODE[23854] := 16#C760;
   // GBK_TO_UNICODE[23855] := 16#8381;
   // GBK_TO_UNICODE[23856] := 16#C761;
   // GBK_TO_UNICODE[23857] := 16#8382;
   // GBK_TO_UNICODE[23858] := 16#C762;
   // GBK_TO_UNICODE[23859] := 16#8383;
   // GBK_TO_UNICODE[23860] := 16#C763;
   // GBK_TO_UNICODE[23861] := 16#8384;
   // GBK_TO_UNICODE[23862] := 16#C764;
   // GBK_TO_UNICODE[23863] := 16#8387;
   // GBK_TO_UNICODE[23864] := 16#C765;
   // GBK_TO_UNICODE[23865] := 16#8388;
   // GBK_TO_UNICODE[23866] := 16#C766;
   // GBK_TO_UNICODE[23867] := 16#838A;
   // GBK_TO_UNICODE[23868] := 16#C767;
   // GBK_TO_UNICODE[23869] := 16#838B;
   // GBK_TO_UNICODE[23870] := 16#C768;
   // GBK_TO_UNICODE[23871] := 16#838C;
   // GBK_TO_UNICODE[23872] := 16#C769;
   // GBK_TO_UNICODE[23873] := 16#838D;
   // GBK_TO_UNICODE[23874] := 16#C76A;
   // GBK_TO_UNICODE[23875] := 16#838F;
   // GBK_TO_UNICODE[23876] := 16#C76B;
   // GBK_TO_UNICODE[23877] := 16#8390;
   // GBK_TO_UNICODE[23878] := 16#C76C;
   // GBK_TO_UNICODE[23879] := 16#8391;
   // GBK_TO_UNICODE[23880] := 16#C76D;
   // GBK_TO_UNICODE[23881] := 16#8394;
   // GBK_TO_UNICODE[23882] := 16#C76E;
   // GBK_TO_UNICODE[23883] := 16#8395;
   // GBK_TO_UNICODE[23884] := 16#C76F;
   // GBK_TO_UNICODE[23885] := 16#8396;
   // GBK_TO_UNICODE[23886] := 16#C770;
   // GBK_TO_UNICODE[23887] := 16#8397;
   // GBK_TO_UNICODE[23888] := 16#C771;
   // GBK_TO_UNICODE[23889] := 16#8399;
   // GBK_TO_UNICODE[23890] := 16#C772;
   // GBK_TO_UNICODE[23891] := 16#839A;
   // GBK_TO_UNICODE[23892] := 16#C773;
   // GBK_TO_UNICODE[23893] := 16#839D;
   // GBK_TO_UNICODE[23894] := 16#C774;
   // GBK_TO_UNICODE[23895] := 16#839F;
   // GBK_TO_UNICODE[23896] := 16#C775;
   // GBK_TO_UNICODE[23897] := 16#83A1;
   // GBK_TO_UNICODE[23898] := 16#C776;
   // GBK_TO_UNICODE[23899] := 16#83A2;
   // GBK_TO_UNICODE[23900] := 16#C777;
   // GBK_TO_UNICODE[23901] := 16#83A3;
   // GBK_TO_UNICODE[23902] := 16#C778;
   // GBK_TO_UNICODE[23903] := 16#83A4;
   // GBK_TO_UNICODE[23904] := 16#C779;
   // GBK_TO_UNICODE[23905] := 16#83A5;
   // GBK_TO_UNICODE[23906] := 16#C77A;
   // GBK_TO_UNICODE[23907] := 16#83A6;
   // GBK_TO_UNICODE[23908] := 16#C77B;
   // GBK_TO_UNICODE[23909] := 16#83A7;
   // GBK_TO_UNICODE[23910] := 16#C77C;
   // GBK_TO_UNICODE[23911] := 16#83AC;
   // GBK_TO_UNICODE[23912] := 16#C77D;
   // GBK_TO_UNICODE[23913] := 16#83AD;
   // GBK_TO_UNICODE[23914] := 16#C77E;
   // GBK_TO_UNICODE[23915] := 16#83AE;
   // GBK_TO_UNICODE[23916] := 16#C780;
   // GBK_TO_UNICODE[23917] := 16#83AF;
   // GBK_TO_UNICODE[23918] := 16#C781;
   // GBK_TO_UNICODE[23919] := 16#83B5;
   // GBK_TO_UNICODE[23920] := 16#C782;
   // GBK_TO_UNICODE[23921] := 16#83BB;
   // GBK_TO_UNICODE[23922] := 16#C783;
   // GBK_TO_UNICODE[23923] := 16#83BE;
   // GBK_TO_UNICODE[23924] := 16#C784;
   // GBK_TO_UNICODE[23925] := 16#83BF;
   // GBK_TO_UNICODE[23926] := 16#C785;
   // GBK_TO_UNICODE[23927] := 16#83C2;
   // GBK_TO_UNICODE[23928] := 16#C786;
   // GBK_TO_UNICODE[23929] := 16#83C3;
   // GBK_TO_UNICODE[23930] := 16#C787;
   // GBK_TO_UNICODE[23931] := 16#83C4;
   // GBK_TO_UNICODE[23932] := 16#C788;
   // GBK_TO_UNICODE[23933] := 16#83C6;
   // GBK_TO_UNICODE[23934] := 16#C789;
   // GBK_TO_UNICODE[23935] := 16#83C8;
   // GBK_TO_UNICODE[23936] := 16#C78A;
   // GBK_TO_UNICODE[23937] := 16#83C9;
   // GBK_TO_UNICODE[23938] := 16#C78B;
   // GBK_TO_UNICODE[23939] := 16#83CB;
   // GBK_TO_UNICODE[23940] := 16#C78C;
   // GBK_TO_UNICODE[23941] := 16#83CD;
   // GBK_TO_UNICODE[23942] := 16#C78D;
   // GBK_TO_UNICODE[23943] := 16#83CE;
   // GBK_TO_UNICODE[23944] := 16#C78E;
   // GBK_TO_UNICODE[23945] := 16#83D0;
   // GBK_TO_UNICODE[23946] := 16#C78F;
   // GBK_TO_UNICODE[23947] := 16#83D1;
   // GBK_TO_UNICODE[23948] := 16#C790;
   // GBK_TO_UNICODE[23949] := 16#83D2;
   // GBK_TO_UNICODE[23950] := 16#C791;
   // GBK_TO_UNICODE[23951] := 16#83D3;
   // GBK_TO_UNICODE[23952] := 16#C792;
   // GBK_TO_UNICODE[23953] := 16#83D5;
   // GBK_TO_UNICODE[23954] := 16#C793;
   // GBK_TO_UNICODE[23955] := 16#83D7;
   // GBK_TO_UNICODE[23956] := 16#C794;
   // GBK_TO_UNICODE[23957] := 16#83D9;
   // GBK_TO_UNICODE[23958] := 16#C795;
   // GBK_TO_UNICODE[23959] := 16#83DA;
   // GBK_TO_UNICODE[23960] := 16#C796;
   // GBK_TO_UNICODE[23961] := 16#83DB;
   // GBK_TO_UNICODE[23962] := 16#C797;
   // GBK_TO_UNICODE[23963] := 16#83DE;
   // GBK_TO_UNICODE[23964] := 16#C798;
   // GBK_TO_UNICODE[23965] := 16#83E2;
   // GBK_TO_UNICODE[23966] := 16#C799;
   // GBK_TO_UNICODE[23967] := 16#83E3;
   // GBK_TO_UNICODE[23968] := 16#C79A;
   // GBK_TO_UNICODE[23969] := 16#83E4;
   // GBK_TO_UNICODE[23970] := 16#C79B;
   // GBK_TO_UNICODE[23971] := 16#83E6;
   // GBK_TO_UNICODE[23972] := 16#C79C;
   // GBK_TO_UNICODE[23973] := 16#83E7;
   // GBK_TO_UNICODE[23974] := 16#C79D;
   // GBK_TO_UNICODE[23975] := 16#83E8;
   // GBK_TO_UNICODE[23976] := 16#C79E;
   // GBK_TO_UNICODE[23977] := 16#83EB;
   // GBK_TO_UNICODE[23978] := 16#C79F;
   // GBK_TO_UNICODE[23979] := 16#83EC;
   // GBK_TO_UNICODE[23980] := 16#C7A0;
   // GBK_TO_UNICODE[23981] := 16#83ED;
   // GBK_TO_UNICODE[23982] := 16#C7A1;
   // GBK_TO_UNICODE[23983] := 16#6070;
   // GBK_TO_UNICODE[23984] := 16#C7A2;
   // GBK_TO_UNICODE[23985] := 16#6D3D;
   // GBK_TO_UNICODE[23986] := 16#C7A3;
   // GBK_TO_UNICODE[23987] := 16#7275;
   // GBK_TO_UNICODE[23988] := 16#C7A4;
   // GBK_TO_UNICODE[23989] := 16#6266;
   // GBK_TO_UNICODE[23990] := 16#C7A5;
   // GBK_TO_UNICODE[23991] := 16#948E;
   // GBK_TO_UNICODE[23992] := 16#C7A6;
   // GBK_TO_UNICODE[23993] := 16#94C5;
   // GBK_TO_UNICODE[23994] := 16#C7A7;
   // GBK_TO_UNICODE[23995] := 16#5343;
   // GBK_TO_UNICODE[23996] := 16#C7A8;
   // GBK_TO_UNICODE[23997] := 16#8FC1;
   // GBK_TO_UNICODE[23998] := 16#C7A9;
   // GBK_TO_UNICODE[23999] := 16#7B7E;
   // GBK_TO_UNICODE[24000] := 16#C7AA;
   // GBK_TO_UNICODE[24001] := 16#4EDF;
   // GBK_TO_UNICODE[24002] := 16#C7AB;
   // GBK_TO_UNICODE[24003] := 16#8C26;
   // GBK_TO_UNICODE[24004] := 16#C7AC;
   // GBK_TO_UNICODE[24005] := 16#4E7E;
   // GBK_TO_UNICODE[24006] := 16#C7AD;
   // GBK_TO_UNICODE[24007] := 16#9ED4;
   // GBK_TO_UNICODE[24008] := 16#C7AE;
   // GBK_TO_UNICODE[24009] := 16#94B1;
   // GBK_TO_UNICODE[24010] := 16#C7AF;
   // GBK_TO_UNICODE[24011] := 16#94B3;
   // GBK_TO_UNICODE[24012] := 16#C7B0;
   // GBK_TO_UNICODE[24013] := 16#524D;
   // GBK_TO_UNICODE[24014] := 16#C7B1;
   // GBK_TO_UNICODE[24015] := 16#6F5C;
   // GBK_TO_UNICODE[24016] := 16#C7B2;
   // GBK_TO_UNICODE[24017] := 16#9063;
   // GBK_TO_UNICODE[24018] := 16#C7B3;
   // GBK_TO_UNICODE[24019] := 16#6D45;
   // GBK_TO_UNICODE[24020] := 16#C7B4;
   // GBK_TO_UNICODE[24021] := 16#8C34;
   // GBK_TO_UNICODE[24022] := 16#C7B5;
   // GBK_TO_UNICODE[24023] := 16#5811;
   // GBK_TO_UNICODE[24024] := 16#C7B6;
   // GBK_TO_UNICODE[24025] := 16#5D4C;
   // GBK_TO_UNICODE[24026] := 16#C7B7;
   // GBK_TO_UNICODE[24027] := 16#6B20;
   // GBK_TO_UNICODE[24028] := 16#C7B8;
   // GBK_TO_UNICODE[24029] := 16#6B49;
   // GBK_TO_UNICODE[24030] := 16#C7B9;
   // GBK_TO_UNICODE[24031] := 16#67AA;
   // GBK_TO_UNICODE[24032] := 16#C7BA;
   // GBK_TO_UNICODE[24033] := 16#545B;
   // GBK_TO_UNICODE[24034] := 16#C7BB;
   // GBK_TO_UNICODE[24035] := 16#8154;
   // GBK_TO_UNICODE[24036] := 16#C7BC;
   // GBK_TO_UNICODE[24037] := 16#7F8C;
   // GBK_TO_UNICODE[24038] := 16#C7BD;
   // GBK_TO_UNICODE[24039] := 16#5899;
   // GBK_TO_UNICODE[24040] := 16#C7BE;
   // GBK_TO_UNICODE[24041] := 16#8537;
   // GBK_TO_UNICODE[24042] := 16#C7BF;
   // GBK_TO_UNICODE[24043] := 16#5F3A;
   // GBK_TO_UNICODE[24044] := 16#C7C0;
   // GBK_TO_UNICODE[24045] := 16#62A2;
   // GBK_TO_UNICODE[24046] := 16#C7C1;
   // GBK_TO_UNICODE[24047] := 16#6A47;
   // GBK_TO_UNICODE[24048] := 16#C7C2;
   // GBK_TO_UNICODE[24049] := 16#9539;
   // GBK_TO_UNICODE[24050] := 16#C7C3;
   // GBK_TO_UNICODE[24051] := 16#6572;
   // GBK_TO_UNICODE[24052] := 16#C7C4;
   // GBK_TO_UNICODE[24053] := 16#6084;
   // GBK_TO_UNICODE[24054] := 16#C7C5;
   // GBK_TO_UNICODE[24055] := 16#6865;
   // GBK_TO_UNICODE[24056] := 16#C7C6;
   // GBK_TO_UNICODE[24057] := 16#77A7;
   // GBK_TO_UNICODE[24058] := 16#C7C7;
   // GBK_TO_UNICODE[24059] := 16#4E54;
   // GBK_TO_UNICODE[24060] := 16#C7C8;
   // GBK_TO_UNICODE[24061] := 16#4FA8;
   // GBK_TO_UNICODE[24062] := 16#C7C9;
   // GBK_TO_UNICODE[24063] := 16#5DE7;
   // GBK_TO_UNICODE[24064] := 16#C7CA;
   // GBK_TO_UNICODE[24065] := 16#9798;
   // GBK_TO_UNICODE[24066] := 16#C7CB;
   // GBK_TO_UNICODE[24067] := 16#64AC;
   // GBK_TO_UNICODE[24068] := 16#C7CC;
   // GBK_TO_UNICODE[24069] := 16#7FD8;
   // GBK_TO_UNICODE[24070] := 16#C7CD;
   // GBK_TO_UNICODE[24071] := 16#5CED;
   // GBK_TO_UNICODE[24072] := 16#C7CE;
   // GBK_TO_UNICODE[24073] := 16#4FCF;
   // GBK_TO_UNICODE[24074] := 16#C7CF;
   // GBK_TO_UNICODE[24075] := 16#7A8D;
   // GBK_TO_UNICODE[24076] := 16#C7D0;
   // GBK_TO_UNICODE[24077] := 16#5207;
   // GBK_TO_UNICODE[24078] := 16#C7D1;
   // GBK_TO_UNICODE[24079] := 16#8304;
   // GBK_TO_UNICODE[24080] := 16#C7D2;
   // GBK_TO_UNICODE[24081] := 16#4E14;
   // GBK_TO_UNICODE[24082] := 16#C7D3;
   // GBK_TO_UNICODE[24083] := 16#602F;
   // GBK_TO_UNICODE[24084] := 16#C7D4;
   // GBK_TO_UNICODE[24085] := 16#7A83;
   // GBK_TO_UNICODE[24086] := 16#C7D5;
   // GBK_TO_UNICODE[24087] := 16#94A6;
   // GBK_TO_UNICODE[24088] := 16#C7D6;
   // GBK_TO_UNICODE[24089] := 16#4FB5;
   // GBK_TO_UNICODE[24090] := 16#C7D7;
   // GBK_TO_UNICODE[24091] := 16#4EB2;
   // GBK_TO_UNICODE[24092] := 16#C7D8;
   // GBK_TO_UNICODE[24093] := 16#79E6;
   // GBK_TO_UNICODE[24094] := 16#C7D9;
   // GBK_TO_UNICODE[24095] := 16#7434;
   // GBK_TO_UNICODE[24096] := 16#C7DA;
   // GBK_TO_UNICODE[24097] := 16#52E4;
   // GBK_TO_UNICODE[24098] := 16#C7DB;
   // GBK_TO_UNICODE[24099] := 16#82B9;
   // GBK_TO_UNICODE[24100] := 16#C7DC;
   // GBK_TO_UNICODE[24101] := 16#64D2;
   // GBK_TO_UNICODE[24102] := 16#C7DD;
   // GBK_TO_UNICODE[24103] := 16#79BD;
   // GBK_TO_UNICODE[24104] := 16#C7DE;
   // GBK_TO_UNICODE[24105] := 16#5BDD;
   // GBK_TO_UNICODE[24106] := 16#C7DF;
   // GBK_TO_UNICODE[24107] := 16#6C81;
   // GBK_TO_UNICODE[24108] := 16#C7E0;
   // GBK_TO_UNICODE[24109] := 16#9752;
   // GBK_TO_UNICODE[24110] := 16#C7E1;
   // GBK_TO_UNICODE[24111] := 16#8F7B;
   // GBK_TO_UNICODE[24112] := 16#C7E2;
   // GBK_TO_UNICODE[24113] := 16#6C22;
   // GBK_TO_UNICODE[24114] := 16#C7E3;
   // GBK_TO_UNICODE[24115] := 16#503E;
   // GBK_TO_UNICODE[24116] := 16#C7E4;
   // GBK_TO_UNICODE[24117] := 16#537F;
   // GBK_TO_UNICODE[24118] := 16#C7E5;
   // GBK_TO_UNICODE[24119] := 16#6E05;
   // GBK_TO_UNICODE[24120] := 16#C7E6;
   // GBK_TO_UNICODE[24121] := 16#64CE;
   // GBK_TO_UNICODE[24122] := 16#C7E7;
   // GBK_TO_UNICODE[24123] := 16#6674;
   // GBK_TO_UNICODE[24124] := 16#C7E8;
   // GBK_TO_UNICODE[24125] := 16#6C30;
   // GBK_TO_UNICODE[24126] := 16#C7E9;
   // GBK_TO_UNICODE[24127] := 16#60C5;
   // GBK_TO_UNICODE[24128] := 16#C7EA;
   // GBK_TO_UNICODE[24129] := 16#9877;
   // GBK_TO_UNICODE[24130] := 16#C7EB;
   // GBK_TO_UNICODE[24131] := 16#8BF7;
   // GBK_TO_UNICODE[24132] := 16#C7EC;
   // GBK_TO_UNICODE[24133] := 16#5E86;
   // GBK_TO_UNICODE[24134] := 16#C7ED;
   // GBK_TO_UNICODE[24135] := 16#743C;
   // GBK_TO_UNICODE[24136] := 16#C7EE;
   // GBK_TO_UNICODE[24137] := 16#7A77;
   // GBK_TO_UNICODE[24138] := 16#C7EF;
   // GBK_TO_UNICODE[24139] := 16#79CB;
   // GBK_TO_UNICODE[24140] := 16#C7F0;
   // GBK_TO_UNICODE[24141] := 16#4E18;
   // GBK_TO_UNICODE[24142] := 16#C7F1;
   // GBK_TO_UNICODE[24143] := 16#90B1;
   // GBK_TO_UNICODE[24144] := 16#C7F2;
   // GBK_TO_UNICODE[24145] := 16#7403;
   // GBK_TO_UNICODE[24146] := 16#C7F3;
   // GBK_TO_UNICODE[24147] := 16#6C42;
   // GBK_TO_UNICODE[24148] := 16#C7F4;
   // GBK_TO_UNICODE[24149] := 16#56DA;
   // GBK_TO_UNICODE[24150] := 16#C7F5;
   // GBK_TO_UNICODE[24151] := 16#914B;
   // GBK_TO_UNICODE[24152] := 16#C7F6;
   // GBK_TO_UNICODE[24153] := 16#6CC5;
   // GBK_TO_UNICODE[24154] := 16#C7F7;
   // GBK_TO_UNICODE[24155] := 16#8D8B;
   // GBK_TO_UNICODE[24156] := 16#C7F8;
   // GBK_TO_UNICODE[24157] := 16#533A;
   // GBK_TO_UNICODE[24158] := 16#C7F9;
   // GBK_TO_UNICODE[24159] := 16#86C6;
   // GBK_TO_UNICODE[24160] := 16#C7FA;
   // GBK_TO_UNICODE[24161] := 16#66F2;
   // GBK_TO_UNICODE[24162] := 16#C7FB;
   // GBK_TO_UNICODE[24163] := 16#8EAF;
   // GBK_TO_UNICODE[24164] := 16#C7FC;
   // GBK_TO_UNICODE[24165] := 16#5C48;
   // GBK_TO_UNICODE[24166] := 16#C7FD;
   // GBK_TO_UNICODE[24167] := 16#9A71;
   // GBK_TO_UNICODE[24168] := 16#C7FE;
   // GBK_TO_UNICODE[24169] := 16#6E20;
   // GBK_TO_UNICODE[24170] := 16#C840;
   // GBK_TO_UNICODE[24171] := 16#83EE;
   // GBK_TO_UNICODE[24172] := 16#C841;
   // GBK_TO_UNICODE[24173] := 16#83EF;
   // GBK_TO_UNICODE[24174] := 16#C842;
   // GBK_TO_UNICODE[24175] := 16#83F3;
   // GBK_TO_UNICODE[24176] := 16#C843;
   // GBK_TO_UNICODE[24177] := 16#83F4;
   // GBK_TO_UNICODE[24178] := 16#C844;
   // GBK_TO_UNICODE[24179] := 16#83F5;
   // GBK_TO_UNICODE[24180] := 16#C845;
   // GBK_TO_UNICODE[24181] := 16#83F6;
   // GBK_TO_UNICODE[24182] := 16#C846;
   // GBK_TO_UNICODE[24183] := 16#83F7;
   // GBK_TO_UNICODE[24184] := 16#C847;
   // GBK_TO_UNICODE[24185] := 16#83FA;
   // GBK_TO_UNICODE[24186] := 16#C848;
   // GBK_TO_UNICODE[24187] := 16#83FB;
   // GBK_TO_UNICODE[24188] := 16#C849;
   // GBK_TO_UNICODE[24189] := 16#83FC;
   // GBK_TO_UNICODE[24190] := 16#C84A;
   // GBK_TO_UNICODE[24191] := 16#83FE;
   // GBK_TO_UNICODE[24192] := 16#C84B;
   // GBK_TO_UNICODE[24193] := 16#83FF;
   // GBK_TO_UNICODE[24194] := 16#C84C;
   // GBK_TO_UNICODE[24195] := 16#8400;
   // GBK_TO_UNICODE[24196] := 16#C84D;
   // GBK_TO_UNICODE[24197] := 16#8402;
   // GBK_TO_UNICODE[24198] := 16#C84E;
   // GBK_TO_UNICODE[24199] := 16#8405;
   // GBK_TO_UNICODE[24200] := 16#C84F;
   // GBK_TO_UNICODE[24201] := 16#8407;
   // GBK_TO_UNICODE[24202] := 16#C850;
   // GBK_TO_UNICODE[24203] := 16#8408;
   // GBK_TO_UNICODE[24204] := 16#C851;
   // GBK_TO_UNICODE[24205] := 16#8409;
   // GBK_TO_UNICODE[24206] := 16#C852;
   // GBK_TO_UNICODE[24207] := 16#840A;
   // GBK_TO_UNICODE[24208] := 16#C853;
   // GBK_TO_UNICODE[24209] := 16#8410;
   // GBK_TO_UNICODE[24210] := 16#C854;
   // GBK_TO_UNICODE[24211] := 16#8412;
   // GBK_TO_UNICODE[24212] := 16#C855;
   // GBK_TO_UNICODE[24213] := 16#8413;
   // GBK_TO_UNICODE[24214] := 16#C856;
   // GBK_TO_UNICODE[24215] := 16#8414;
   // GBK_TO_UNICODE[24216] := 16#C857;
   // GBK_TO_UNICODE[24217] := 16#8415;
   // GBK_TO_UNICODE[24218] := 16#C858;
   // GBK_TO_UNICODE[24219] := 16#8416;
   // GBK_TO_UNICODE[24220] := 16#C859;
   // GBK_TO_UNICODE[24221] := 16#8417;
   // GBK_TO_UNICODE[24222] := 16#C85A;
   // GBK_TO_UNICODE[24223] := 16#8419;
   // GBK_TO_UNICODE[24224] := 16#C85B;
   // GBK_TO_UNICODE[24225] := 16#841A;
   // GBK_TO_UNICODE[24226] := 16#C85C;
   // GBK_TO_UNICODE[24227] := 16#841B;
   // GBK_TO_UNICODE[24228] := 16#C85D;
   // GBK_TO_UNICODE[24229] := 16#841E;
   // GBK_TO_UNICODE[24230] := 16#C85E;
   // GBK_TO_UNICODE[24231] := 16#841F;
   // GBK_TO_UNICODE[24232] := 16#C85F;
   // GBK_TO_UNICODE[24233] := 16#8420;
   // GBK_TO_UNICODE[24234] := 16#C860;
   // GBK_TO_UNICODE[24235] := 16#8421;
   // GBK_TO_UNICODE[24236] := 16#C861;
   // GBK_TO_UNICODE[24237] := 16#8422;
   // GBK_TO_UNICODE[24238] := 16#C862;
   // GBK_TO_UNICODE[24239] := 16#8423;
   // GBK_TO_UNICODE[24240] := 16#C863;
   // GBK_TO_UNICODE[24241] := 16#8429;
   // GBK_TO_UNICODE[24242] := 16#C864;
   // GBK_TO_UNICODE[24243] := 16#842A;
   // GBK_TO_UNICODE[24244] := 16#C865;
   // GBK_TO_UNICODE[24245] := 16#842B;
   // GBK_TO_UNICODE[24246] := 16#C866;
   // GBK_TO_UNICODE[24247] := 16#842C;
   // GBK_TO_UNICODE[24248] := 16#C867;
   // GBK_TO_UNICODE[24249] := 16#842D;
   // GBK_TO_UNICODE[24250] := 16#C868;
   // GBK_TO_UNICODE[24251] := 16#842E;
   // GBK_TO_UNICODE[24252] := 16#C869;
   // GBK_TO_UNICODE[24253] := 16#842F;
   // GBK_TO_UNICODE[24254] := 16#C86A;
   // GBK_TO_UNICODE[24255] := 16#8430;
   // GBK_TO_UNICODE[24256] := 16#C86B;
   // GBK_TO_UNICODE[24257] := 16#8432;
   // GBK_TO_UNICODE[24258] := 16#C86C;
   // GBK_TO_UNICODE[24259] := 16#8433;
   // GBK_TO_UNICODE[24260] := 16#C86D;
   // GBK_TO_UNICODE[24261] := 16#8434;
   // GBK_TO_UNICODE[24262] := 16#C86E;
   // GBK_TO_UNICODE[24263] := 16#8435;
   // GBK_TO_UNICODE[24264] := 16#C86F;
   // GBK_TO_UNICODE[24265] := 16#8436;
   // GBK_TO_UNICODE[24266] := 16#C870;
   // GBK_TO_UNICODE[24267] := 16#8437;
   // GBK_TO_UNICODE[24268] := 16#C871;
   // GBK_TO_UNICODE[24269] := 16#8439;
   // GBK_TO_UNICODE[24270] := 16#C872;
   // GBK_TO_UNICODE[24271] := 16#843A;
   // GBK_TO_UNICODE[24272] := 16#C873;
   // GBK_TO_UNICODE[24273] := 16#843B;
   // GBK_TO_UNICODE[24274] := 16#C874;
   // GBK_TO_UNICODE[24275] := 16#843E;
   // GBK_TO_UNICODE[24276] := 16#C875;
   // GBK_TO_UNICODE[24277] := 16#843F;
   // GBK_TO_UNICODE[24278] := 16#C876;
   // GBK_TO_UNICODE[24279] := 16#8440;
   // GBK_TO_UNICODE[24280] := 16#C877;
   // GBK_TO_UNICODE[24281] := 16#8441;
   // GBK_TO_UNICODE[24282] := 16#C878;
   // GBK_TO_UNICODE[24283] := 16#8442;
   // GBK_TO_UNICODE[24284] := 16#C879;
   // GBK_TO_UNICODE[24285] := 16#8443;
   // GBK_TO_UNICODE[24286] := 16#C87A;
   // GBK_TO_UNICODE[24287] := 16#8444;
   // GBK_TO_UNICODE[24288] := 16#C87B;
   // GBK_TO_UNICODE[24289] := 16#8445;
   // GBK_TO_UNICODE[24290] := 16#C87C;
   // GBK_TO_UNICODE[24291] := 16#8447;
   // GBK_TO_UNICODE[24292] := 16#C87D;
   // GBK_TO_UNICODE[24293] := 16#8448;
   // GBK_TO_UNICODE[24294] := 16#C87E;
   // GBK_TO_UNICODE[24295] := 16#8449;
   // GBK_TO_UNICODE[24296] := 16#C880;
   // GBK_TO_UNICODE[24297] := 16#844A;
   // GBK_TO_UNICODE[24298] := 16#C881;
   // GBK_TO_UNICODE[24299] := 16#844B;
   // GBK_TO_UNICODE[24300] := 16#C882;
   // GBK_TO_UNICODE[24301] := 16#844C;
   // GBK_TO_UNICODE[24302] := 16#C883;
   // GBK_TO_UNICODE[24303] := 16#844D;
   // GBK_TO_UNICODE[24304] := 16#C884;
   // GBK_TO_UNICODE[24305] := 16#844E;
   // GBK_TO_UNICODE[24306] := 16#C885;
   // GBK_TO_UNICODE[24307] := 16#844F;
   // GBK_TO_UNICODE[24308] := 16#C886;
   // GBK_TO_UNICODE[24309] := 16#8450;
   // GBK_TO_UNICODE[24310] := 16#C887;
   // GBK_TO_UNICODE[24311] := 16#8452;
   // GBK_TO_UNICODE[24312] := 16#C888;
   // GBK_TO_UNICODE[24313] := 16#8453;
   // GBK_TO_UNICODE[24314] := 16#C889;
   // GBK_TO_UNICODE[24315] := 16#8454;
   // GBK_TO_UNICODE[24316] := 16#C88A;
   // GBK_TO_UNICODE[24317] := 16#8455;
   // GBK_TO_UNICODE[24318] := 16#C88B;
   // GBK_TO_UNICODE[24319] := 16#8456;
   // GBK_TO_UNICODE[24320] := 16#C88C;
   // GBK_TO_UNICODE[24321] := 16#8458;
   // GBK_TO_UNICODE[24322] := 16#C88D;
   // GBK_TO_UNICODE[24323] := 16#845D;
   // GBK_TO_UNICODE[24324] := 16#C88E;
   // GBK_TO_UNICODE[24325] := 16#845E;
   // GBK_TO_UNICODE[24326] := 16#C88F;
   // GBK_TO_UNICODE[24327] := 16#845F;
   // GBK_TO_UNICODE[24328] := 16#C890;
   // GBK_TO_UNICODE[24329] := 16#8460;
   // GBK_TO_UNICODE[24330] := 16#C891;
   // GBK_TO_UNICODE[24331] := 16#8462;
   // GBK_TO_UNICODE[24332] := 16#C892;
   // GBK_TO_UNICODE[24333] := 16#8464;
   // GBK_TO_UNICODE[24334] := 16#C893;
   // GBK_TO_UNICODE[24335] := 16#8465;
   // GBK_TO_UNICODE[24336] := 16#C894;
   // GBK_TO_UNICODE[24337] := 16#8466;
   // GBK_TO_UNICODE[24338] := 16#C895;
   // GBK_TO_UNICODE[24339] := 16#8467;
   // GBK_TO_UNICODE[24340] := 16#C896;
   // GBK_TO_UNICODE[24341] := 16#8468;
   // GBK_TO_UNICODE[24342] := 16#C897;
   // GBK_TO_UNICODE[24343] := 16#846A;
   // GBK_TO_UNICODE[24344] := 16#C898;
   // GBK_TO_UNICODE[24345] := 16#846E;
   // GBK_TO_UNICODE[24346] := 16#C899;
   // GBK_TO_UNICODE[24347] := 16#846F;
   // GBK_TO_UNICODE[24348] := 16#C89A;
   // GBK_TO_UNICODE[24349] := 16#8470;
   // GBK_TO_UNICODE[24350] := 16#C89B;
   // GBK_TO_UNICODE[24351] := 16#8472;
   // GBK_TO_UNICODE[24352] := 16#C89C;
   // GBK_TO_UNICODE[24353] := 16#8474;
   // GBK_TO_UNICODE[24354] := 16#C89D;
   // GBK_TO_UNICODE[24355] := 16#8477;
   // GBK_TO_UNICODE[24356] := 16#C89E;
   // GBK_TO_UNICODE[24357] := 16#8479;
   // GBK_TO_UNICODE[24358] := 16#C89F;
   // GBK_TO_UNICODE[24359] := 16#847B;
   // GBK_TO_UNICODE[24360] := 16#C8A0;
   // GBK_TO_UNICODE[24361] := 16#847C;
   // GBK_TO_UNICODE[24362] := 16#C8A1;
   // GBK_TO_UNICODE[24363] := 16#53D6;
   // GBK_TO_UNICODE[24364] := 16#C8A2;
   // GBK_TO_UNICODE[24365] := 16#5A36;
   // GBK_TO_UNICODE[24366] := 16#C8A3;
   // GBK_TO_UNICODE[24367] := 16#9F8B;
   // GBK_TO_UNICODE[24368] := 16#C8A4;
   // GBK_TO_UNICODE[24369] := 16#8DA3;
   // GBK_TO_UNICODE[24370] := 16#C8A5;
   // GBK_TO_UNICODE[24371] := 16#53BB;
   // GBK_TO_UNICODE[24372] := 16#C8A6;
   // GBK_TO_UNICODE[24373] := 16#5708;
   // GBK_TO_UNICODE[24374] := 16#C8A7;
   // GBK_TO_UNICODE[24375] := 16#98A7;
   // GBK_TO_UNICODE[24376] := 16#C8A8;
   // GBK_TO_UNICODE[24377] := 16#6743;
   // GBK_TO_UNICODE[24378] := 16#C8A9;
   // GBK_TO_UNICODE[24379] := 16#919B;
   // GBK_TO_UNICODE[24380] := 16#C8AA;
   // GBK_TO_UNICODE[24381] := 16#6CC9;
   // GBK_TO_UNICODE[24382] := 16#C8AB;
   // GBK_TO_UNICODE[24383] := 16#5168;
   // GBK_TO_UNICODE[24384] := 16#C8AC;
   // GBK_TO_UNICODE[24385] := 16#75CA;
   // GBK_TO_UNICODE[24386] := 16#C8AD;
   // GBK_TO_UNICODE[24387] := 16#62F3;
   // GBK_TO_UNICODE[24388] := 16#C8AE;
   // GBK_TO_UNICODE[24389] := 16#72AC;
   // GBK_TO_UNICODE[24390] := 16#C8AF;
   // GBK_TO_UNICODE[24391] := 16#5238;
   // GBK_TO_UNICODE[24392] := 16#C8B0;
   // GBK_TO_UNICODE[24393] := 16#529D;
   // GBK_TO_UNICODE[24394] := 16#C8B1;
   // GBK_TO_UNICODE[24395] := 16#7F3A;
   // GBK_TO_UNICODE[24396] := 16#C8B2;
   // GBK_TO_UNICODE[24397] := 16#7094;
   // GBK_TO_UNICODE[24398] := 16#C8B3;
   // GBK_TO_UNICODE[24399] := 16#7638;
   // GBK_TO_UNICODE[24400] := 16#C8B4;
   // GBK_TO_UNICODE[24401] := 16#5374;
   // GBK_TO_UNICODE[24402] := 16#C8B5;
   // GBK_TO_UNICODE[24403] := 16#9E4A;
   // GBK_TO_UNICODE[24404] := 16#C8B6;
   // GBK_TO_UNICODE[24405] := 16#69B7;
   // GBK_TO_UNICODE[24406] := 16#C8B7;
   // GBK_TO_UNICODE[24407] := 16#786E;
   // GBK_TO_UNICODE[24408] := 16#C8B8;
   // GBK_TO_UNICODE[24409] := 16#96C0;
   // GBK_TO_UNICODE[24410] := 16#C8B9;
   // GBK_TO_UNICODE[24411] := 16#88D9;
   // GBK_TO_UNICODE[24412] := 16#C8BA;
   // GBK_TO_UNICODE[24413] := 16#7FA4;
   // GBK_TO_UNICODE[24414] := 16#C8BB;
   // GBK_TO_UNICODE[24415] := 16#7136;
   // GBK_TO_UNICODE[24416] := 16#C8BC;
   // GBK_TO_UNICODE[24417] := 16#71C3;
   // GBK_TO_UNICODE[24418] := 16#C8BD;
   // GBK_TO_UNICODE[24419] := 16#5189;
   // GBK_TO_UNICODE[24420] := 16#C8BE;
   // GBK_TO_UNICODE[24421] := 16#67D3;
   // GBK_TO_UNICODE[24422] := 16#C8BF;
   // GBK_TO_UNICODE[24423] := 16#74E4;
   // GBK_TO_UNICODE[24424] := 16#C8C0;
   // GBK_TO_UNICODE[24425] := 16#58E4;
   // GBK_TO_UNICODE[24426] := 16#C8C1;
   // GBK_TO_UNICODE[24427] := 16#6518;
   // GBK_TO_UNICODE[24428] := 16#C8C2;
   // GBK_TO_UNICODE[24429] := 16#56B7;
   // GBK_TO_UNICODE[24430] := 16#C8C3;
   // GBK_TO_UNICODE[24431] := 16#8BA9;
   // GBK_TO_UNICODE[24432] := 16#C8C4;
   // GBK_TO_UNICODE[24433] := 16#9976;
   // GBK_TO_UNICODE[24434] := 16#C8C5;
   // GBK_TO_UNICODE[24435] := 16#6270;
   // GBK_TO_UNICODE[24436] := 16#C8C6;
   // GBK_TO_UNICODE[24437] := 16#7ED5;
   // GBK_TO_UNICODE[24438] := 16#C8C7;
   // GBK_TO_UNICODE[24439] := 16#60F9;
   // GBK_TO_UNICODE[24440] := 16#C8C8;
   // GBK_TO_UNICODE[24441] := 16#70ED;
   // GBK_TO_UNICODE[24442] := 16#C8C9;
   // GBK_TO_UNICODE[24443] := 16#58EC;
   // GBK_TO_UNICODE[24444] := 16#C8CA;
   // GBK_TO_UNICODE[24445] := 16#4EC1;
   // GBK_TO_UNICODE[24446] := 16#C8CB;
   // GBK_TO_UNICODE[24447] := 16#4EBA;
   // GBK_TO_UNICODE[24448] := 16#C8CC;
   // GBK_TO_UNICODE[24449] := 16#5FCD;
   // GBK_TO_UNICODE[24450] := 16#C8CD;
   // GBK_TO_UNICODE[24451] := 16#97E7;
   // GBK_TO_UNICODE[24452] := 16#C8CE;
   // GBK_TO_UNICODE[24453] := 16#4EFB;
   // GBK_TO_UNICODE[24454] := 16#C8CF;
   // GBK_TO_UNICODE[24455] := 16#8BA4;
   // GBK_TO_UNICODE[24456] := 16#C8D0;
   // GBK_TO_UNICODE[24457] := 16#5203;
   // GBK_TO_UNICODE[24458] := 16#C8D1;
   // GBK_TO_UNICODE[24459] := 16#598A;
   // GBK_TO_UNICODE[24460] := 16#C8D2;
   // GBK_TO_UNICODE[24461] := 16#7EAB;
   // GBK_TO_UNICODE[24462] := 16#C8D3;
   // GBK_TO_UNICODE[24463] := 16#6254;
   // GBK_TO_UNICODE[24464] := 16#C8D4;
   // GBK_TO_UNICODE[24465] := 16#4ECD;
   // GBK_TO_UNICODE[24466] := 16#C8D5;
   // GBK_TO_UNICODE[24467] := 16#65E5;
   // GBK_TO_UNICODE[24468] := 16#C8D6;
   // GBK_TO_UNICODE[24469] := 16#620E;
   // GBK_TO_UNICODE[24470] := 16#C8D7;
   // GBK_TO_UNICODE[24471] := 16#8338;
   // GBK_TO_UNICODE[24472] := 16#C8D8;
   // GBK_TO_UNICODE[24473] := 16#84C9;
   // GBK_TO_UNICODE[24474] := 16#C8D9;
   // GBK_TO_UNICODE[24475] := 16#8363;
   // GBK_TO_UNICODE[24476] := 16#C8DA;
   // GBK_TO_UNICODE[24477] := 16#878D;
   // GBK_TO_UNICODE[24478] := 16#C8DB;
   // GBK_TO_UNICODE[24479] := 16#7194;
   // GBK_TO_UNICODE[24480] := 16#C8DC;
   // GBK_TO_UNICODE[24481] := 16#6EB6;
   // GBK_TO_UNICODE[24482] := 16#C8DD;
   // GBK_TO_UNICODE[24483] := 16#5BB9;
   // GBK_TO_UNICODE[24484] := 16#C8DE;
   // GBK_TO_UNICODE[24485] := 16#7ED2;
   // GBK_TO_UNICODE[24486] := 16#C8DF;
   // GBK_TO_UNICODE[24487] := 16#5197;
   // GBK_TO_UNICODE[24488] := 16#C8E0;
   // GBK_TO_UNICODE[24489] := 16#63C9;
   // GBK_TO_UNICODE[24490] := 16#C8E1;
   // GBK_TO_UNICODE[24491] := 16#67D4;
   // GBK_TO_UNICODE[24492] := 16#C8E2;
   // GBK_TO_UNICODE[24493] := 16#8089;
   // GBK_TO_UNICODE[24494] := 16#C8E3;
   // GBK_TO_UNICODE[24495] := 16#8339;
   // GBK_TO_UNICODE[24496] := 16#C8E4;
   // GBK_TO_UNICODE[24497] := 16#8815;
   // GBK_TO_UNICODE[24498] := 16#C8E5;
   // GBK_TO_UNICODE[24499] := 16#5112;
   // GBK_TO_UNICODE[24500] := 16#C8E6;
   // GBK_TO_UNICODE[24501] := 16#5B7A;
   // GBK_TO_UNICODE[24502] := 16#C8E7;
   // GBK_TO_UNICODE[24503] := 16#5982;
   // GBK_TO_UNICODE[24504] := 16#C8E8;
   // GBK_TO_UNICODE[24505] := 16#8FB1;
   // GBK_TO_UNICODE[24506] := 16#C8E9;
   // GBK_TO_UNICODE[24507] := 16#4E73;
   // GBK_TO_UNICODE[24508] := 16#C8EA;
   // GBK_TO_UNICODE[24509] := 16#6C5D;
   // GBK_TO_UNICODE[24510] := 16#C8EB;
   // GBK_TO_UNICODE[24511] := 16#5165;
   // GBK_TO_UNICODE[24512] := 16#C8EC;
   // GBK_TO_UNICODE[24513] := 16#8925;
   // GBK_TO_UNICODE[24514] := 16#C8ED;
   // GBK_TO_UNICODE[24515] := 16#8F6F;
   // GBK_TO_UNICODE[24516] := 16#C8EE;
   // GBK_TO_UNICODE[24517] := 16#962E;
   // GBK_TO_UNICODE[24518] := 16#C8EF;
   // GBK_TO_UNICODE[24519] := 16#854A;
   // GBK_TO_UNICODE[24520] := 16#C8F0;
   // GBK_TO_UNICODE[24521] := 16#745E;
   // GBK_TO_UNICODE[24522] := 16#C8F1;
   // GBK_TO_UNICODE[24523] := 16#9510;
   // GBK_TO_UNICODE[24524] := 16#C8F2;
   // GBK_TO_UNICODE[24525] := 16#95F0;
   // GBK_TO_UNICODE[24526] := 16#C8F3;
   // GBK_TO_UNICODE[24527] := 16#6DA6;
   // GBK_TO_UNICODE[24528] := 16#C8F4;
   // GBK_TO_UNICODE[24529] := 16#82E5;
   // GBK_TO_UNICODE[24530] := 16#C8F5;
   // GBK_TO_UNICODE[24531] := 16#5F31;
   // GBK_TO_UNICODE[24532] := 16#C8F6;
   // GBK_TO_UNICODE[24533] := 16#6492;
   // GBK_TO_UNICODE[24534] := 16#C8F7;
   // GBK_TO_UNICODE[24535] := 16#6D12;
   // GBK_TO_UNICODE[24536] := 16#C8F8;
   // GBK_TO_UNICODE[24537] := 16#8428;
   // GBK_TO_UNICODE[24538] := 16#C8F9;
   // GBK_TO_UNICODE[24539] := 16#816E;
   // GBK_TO_UNICODE[24540] := 16#C8FA;
   // GBK_TO_UNICODE[24541] := 16#9CC3;
   // GBK_TO_UNICODE[24542] := 16#C8FB;
   // GBK_TO_UNICODE[24543] := 16#585E;
   // GBK_TO_UNICODE[24544] := 16#C8FC;
   // GBK_TO_UNICODE[24545] := 16#8D5B;
   // GBK_TO_UNICODE[24546] := 16#C8FD;
   // GBK_TO_UNICODE[24547] := 16#4E09;
   // GBK_TO_UNICODE[24548] := 16#C8FE;
   // GBK_TO_UNICODE[24549] := 16#53C1;
   // GBK_TO_UNICODE[24550] := 16#C940;
   // GBK_TO_UNICODE[24551] := 16#847D;
   // GBK_TO_UNICODE[24552] := 16#C941;
   // GBK_TO_UNICODE[24553] := 16#847E;
   // GBK_TO_UNICODE[24554] := 16#C942;
   // GBK_TO_UNICODE[24555] := 16#847F;
   // GBK_TO_UNICODE[24556] := 16#C943;
   // GBK_TO_UNICODE[24557] := 16#8480;
   // GBK_TO_UNICODE[24558] := 16#C944;
   // GBK_TO_UNICODE[24559] := 16#8481;
   // GBK_TO_UNICODE[24560] := 16#C945;
   // GBK_TO_UNICODE[24561] := 16#8483;
   // GBK_TO_UNICODE[24562] := 16#C946;
   // GBK_TO_UNICODE[24563] := 16#8484;
   // GBK_TO_UNICODE[24564] := 16#C947;
   // GBK_TO_UNICODE[24565] := 16#8485;
   // GBK_TO_UNICODE[24566] := 16#C948;
   // GBK_TO_UNICODE[24567] := 16#8486;
